LIN {X 0,Y 372.222,Z 970.071,A -85,B 0,C 180,E1 15608.829,E2 15608.829} C_VEL
LIN {X 0,Y 365.379,Z 983.592,A -85,B 0,C 180,E1 15606.041,E2 15606.041} C_VEL
LIN {X 0,Y 359.083,Z 996.112,A -85,B 0,C 180,E1 15603.054,E2 15603.054} C_VEL
LIN {X 0,Y 352.099,Z 1010.25,A -85,B 0,C 180,E1 15599.052,E2 15599.052} C_VEL
LIN {X 0,Y 347.306,Z 1020.442,A -85,B 0,C 180,E1 15595.585,E2 15595.585} C_VEL
LIN {X 0,Y 343.315,Z 1029.671,A -85,B 0,C 180,E1 15591.888,E2 15591.888} C_VEL
LIN {X 0,Y 339.875,Z 1038.664,A -85,B 0,C 180,E1 15587.462,E2 15587.462} C_VEL
LIN {X 0,Y 337.952,Z 1044.795,A -85,B 0,C 180,E1 15583.691,E2 15583.691} C_VEL
LIN {X 0,Y 336.82,Z 1049.482,A -85,B 0,C 180,E1 15580.087,E2 15580.087} C_VEL
LIN {X 0,Y 336.14,Z 1053.645,A -85,B 0,C 180,E1 15575.805,E2 15575.805} C_VEL
LIN {X 0,Y 335.934,Z 1055.971,A -85,B 0,C 180,E1 15571.876,E2 15571.876} C_VEL
LIN {X 0,Y 335.909,Z 1056.968,A -85,B 0,C 180,E1 15568.635,E2 15568.635} C_VEL
LIN {X 0,Y 335.91,Z 1057.084,A -85,B 0,C 180,E1 15565.39,E2 15565.39} C_VEL
LIN {X 0,Y 335.94,Z 1056.315,A -85,B 0,C 180,E1 15562.131,E2 15562.131} C_VEL
LIN {X 0,Y 336.1,Z 1054.654,A -85,B 0,C 180,E1 15558.85,E2 15558.85} C_VEL
LIN {X 0,Y 336.529,Z 1051.925,A -85,B 0,C 180,E1 15555.372,E2 15555.372} C_VEL
LIN {X 0,Y 337.552,Z 1047.758,A -85,B 0,C 180,E1 15551.521,E2 15551.521} C_VEL
LIN {X 0,Y 339.699,Z 1041.098,A -85,B 0,C 180,E1 15546.953,E2 15546.953} C_VEL
LIN {X 0,Y 342.404,Z 1034.312,A -85,B 0,C 180,E1 15543.275,E2 15543.275} C_VEL
LIN {X 0,Y 346.076,Z 1026.246,A -85,B 0,C 180,E1 15539.628,E2 15539.628} C_VEL
LIN {X 0,Y 352.06,Z 1014.26,A -85,B 0,C 180,E1 15535.19,E2 15535.19} C_VEL
LIN {X 0,Y 357.776,Z 1003.409,A -85,B 0,C 180,E1 15531.856,E2 15531.856} C_VEL
LIN {X 0,Y 365.253,Z 989.805,A -85,B 0,C 180,E1 15528.301,E2 15528.301} C_VEL
LIN {X 0,Y 368.811,Z 983.139,A -85,B 0,C 180,E1 15526.799,E2 15526.799} C_VEL
LIN {X 0,Y 370.327,Z 979.107,A -85,B 0,C 180,E1 15525.802,E2 15525.802} C_VEL
LIN {X 0,Y 371.602,Z 968.39,A -85,B 0,C 180,E1 15522.974,E2 15522.974} C_VEL
LIN {X 0,Y 373.172,Z 964.471,A -85,B 0,C 180,E1 15522.181,E2 15522.181} C_VEL
LIN {X 0,Y 381.333,Z 949.488,A -85,B 0,C 180,E1 15519.689,E2 15519.689} C_VEL
LIN {X 0,Y 390.212,Z 932.645,A -85,B 0,C 180,E1 15517.285,E2 15517.285} C_VEL
LIN {X 0,Y 400.258,Z 912.27,A -85,B 0,C 180,E1 15514.852,E2 15514.852} C_VEL
LIN {X 0,Y 408.245,Z 894.982,A -85,B 0,C 180,E1 15513.106,E2 15513.106} C_VEL
LIN {X 0,Y 416.573,Z 875.657,A -85,B 0,C 180,E1 15511.428,E2 15511.428} C_VEL
LIN {X 0,Y 425.589,Z 852.408,A -85,B 0,C 180,E1 15509.747,E2 15509.747} C_VEL
LIN {X 0,Y 432.181,Z 833.489,A -85,B 0,C 180,E1 15508.598,E2 15508.598} C_VEL
LIN {X 0,Y 438.616,Z 812.853,A -85,B 0,C 180,E1 15507.529,E2 15507.529} C_VEL
LIN {X 0,Y 445.749,Z 786.165,A -85,B 0,C 180,E1 15506.41,E2 15506.41} C_VEL
LIN {X 0,Y 450.602,Z 764.172,A -85,B 0,C 180,E1 15505.676,E2 15505.676} C_VEL
LIN {X 0,Y 454.876,Z 740.778,A -85,B 0,C 180,E1 15505.063,E2 15505.063} C_VEL
LIN {X 0,Y 458.362,Z 713.784,A -85,B 0,C 180,E1 15504.527,E2 15504.527} C_VEL
LIN {X 0,Y 473.41,Z 521.073,A -85,B 0,C 180,E1 15501.495,E2 15501.495} C_VEL
LIN {X 0,Y 477.59,Z 467.874,A -85,B 0,C 180,E1 15500.657,E2 15500.657} C_VEL
LIN {X 0,Y 470.268,Z 455.931,A -85,B 0,C 180,E1 15497.829,E2 15497.829} C_VEL
LIN {X 0,Y 464.119,Z 446.543,A -85,B 0,C 180,E1 15495.047,E2 15495.047} C_VEL
LIN {X 0,Y 460.67,Z 441.475,A -85,B 0,C 180,E1 15493.238,E2 15493.238} C_VEL
LIN {X 0,Y 457.903,Z 437.421,A -85,B 0,C 180,E1 15491.589,E2 15491.589} C_VEL
LIN {X 0,Y 454.898,Z 432.925,A -85,B 0,C 180,E1 15489.489,E2 15489.489} C_VEL
LIN {X 0,Y 451.914,Z 428.441,A -85,B 0,C 180,E1 15486.862,E2 15486.862} C_VEL
LIN {X 0,Y 448.733,Z 423.885,A -85,B 0,C 180,E1 15482.426,E2 15482.426} C_VEL
LIN {X 0,Y 448.35,Z 422.762,A -85,B 0,C 180,E1 15481.278,E2 15481.278} C_VEL
LIN {X 0,Y 448.16,Z 422.66,A -85,B 0,C 180,E1 15476.418,E2 15476.418} C_VEL
LIN {X 0,Y 448.576,Z 423.232,A -85,B 0,C 180,E1 15475.141,E2 15475.141} C_VEL
LIN {X 0,Y 450.853,Z 427.461,A -85,B 0,C 180,E1 15471.326,E2 15471.326} C_VEL
LIN {X 0,Y 452.07,Z 428.734,A -85,B 0,C 180,E1 15470.066,E2 15470.066} C_VEL
LIN {X 0,Y 455.617,Z 434.006,A -85,B 0,C 180,E1 15467.065,E2 15467.065} C_VEL
LIN {X 0,Y 459.489,Z 439.662,A -85,B 0,C 180,E1 15464.54,E2 15464.54} C_VEL
LIN {X 0,Y 462.897,Z 444.822,A -85,B 0,C 180,E1 15462.657,E2 15462.657} C_VEL
LIN {X 0,Y 467.926,Z 452.369,A -85,B 0,C 180,E1 15460.268,E2 15460.268} C_VEL
LIN {X 0,Y 473.578,Z 462.229,A -85,B 0,C 180,E1 15457.892,E2 15457.892} C_VEL
LIN {X 0,Y 477.55,Z 469.616,A -85,B 0,C 180,E1 15456.38,E2 15456.38} C_VEL
LIN {X 0,Y 459.798,Z 699.014,A -85,B 0,C 180,E1 15452.792,E2 15452.792} C_VEL
LIN {X 0,Y 456.746,Z 730.026,A -85,B 0,C 180,E1 15452.255,E2 15452.255} C_VEL
LIN {X 0,Y 453.419,Z 751.939,A -85,B 0,C 180,E1 15451.778,E2 15451.778} C_VEL
LIN {X 0,Y 448.791,Z 775.796,A -85,B 0,C 180,E1 15451.123,E2 15451.123} C_VEL
LIN {X 0,Y 442.754,Z 800.711,A -85,B 0,C 180,E1 15450.229,E2 15450.229} C_VEL
LIN {X 0,Y 436.754,Z 821.884,A -85,B 0,C 180,E1 15449.29,E2 15449.29} C_VEL
LIN {X 0,Y 429.461,Z 844.642,A -85,B 0,C 180,E1 15448.077,E2 15448.077} C_VEL
LIN {X 0,Y 421,Z 867.55,A -85,B 0,C 180,E1 15446.585,E2 15446.585} C_VEL
LIN {X 0,Y 413.553,Z 885.936,A -85,B 0,C 180,E1 15445.169,E2 15445.169} C_VEL
LIN {X 0,Y 404.883,Z 905.797,A -85,B 0,C 180,E1 15443.38,E2 15443.38} C_VEL
LIN {X 0,Y 395.21,Z 926.087,A -85,B 0,C 180,E1 15441.191,E2 15441.191} C_VEL
LIN {X 0,Y 387.162,Z 942.019,A -85,B 0,C 180,E1 15439.174,E2 15439.174} C_VEL
LIN {X 0,Y 378.632,Z 958.248,A -85,B 0,C 180,E1 15436.791,E2 15436.791} C_VEL
LIN {X 0,Y 368.644,Z 976.469,A -85,B 0,C 180,E1 15433.598,E2 15433.598} C_VEL
LIN {X 0,Y 361.117,Z 989.91,A -85,B 0,C 180,E1 15430.802,E2 15430.802} C_VEL
LIN {X 0,Y 353.453,Z 1003.67,A -85,B 0,C 180,E1 15427.461,E2 15427.461} C_VEL
LIN {X 0,Y 346.006,Z 1017.147,A -85,B 0,C 180,E1 15423.501,E2 15423.501} C_VEL
LIN {X 0,Y 340.806,Z 1027.013,A -85,B 0,C 180,E1 15420.06,E2 15420.06} C_VEL
LIN {X 0,Y 335.835,Z 1037.363,A -85,B 0,C 180,E1 15415.765,E2 15415.765} C_VEL
LIN {X 0,Y 332.319,Z 1045.488,A -85,B 0,C 180,E1 15411.535,E2 15411.535} C_VEL
LIN {X 0,Y 330.223,Z 1051.354,A -85,B 0,C 180,E1 15407.807,E2 15407.807} C_VEL
LIN {X 0,Y 328.785,Z 1056.688,A -85,B 0,C 180,E1 15403.543,E2 15403.543} C_VEL
LIN {X 0,Y 328.091,Z 1060.541,A -85,B 0,C 180,E1 15399.095,E2 15399.095} C_VEL
LIN {X 0,Y 327.924,Z 1062.495,A -85,B 0,C 180,E1 15395.599,E2 15395.599} C_VEL
LIN {X 0,Y 327.91,Z 1063.451,A -85,B 0,C 180,E1 15392.272,E2 15392.272} C_VEL
LIN {X 0,Y 327.914,Z 1063.508,A -85,B 0,C 180,E1 15388.952,E2 15388.952} C_VEL
LIN {X 0,Y 327.909,Z 1062.672,A -85,B 0,C 180,E1 15385.652,E2 15385.652} C_VEL
LIN {X 0,Y 328.019,Z 1060.834,A -85,B 0,C 180,E1 15382.177,E2 15382.177} C_VEL
LIN {X 0,Y 328.377,Z 1057.75,A -85,B 0,C 180,E1 15378.407,E2 15378.407} C_VEL
LIN {X 0,Y 329.528,Z 1052.362,A -85,B 0,C 180,E1 15373.79,E2 15373.79} C_VEL
LIN {X 0,Y 331.318,Z 1046.309,A -85,B 0,C 180,E1 15369.877,E2 15369.877} C_VEL
LIN {X 0,Y 333.901,Z 1039.288,A -85,B 0,C 180,E1 15366.155,E2 15366.155} C_VEL
LIN {X 0,Y 338.231,Z 1029.2,A -85,B 0,C 180,E1 15361.759,E2 15361.759} C_VEL
LIN {X 0,Y 343.228,Z 1018.544,A -85,B 0,C 180,E1 15357.967,E2 15357.967} C_VEL
LIN {X 0,Y 348.774,Z 1007.481,A -85,B 0,C 180,E1 15354.613,E2 15354.613} C_VEL
LIN {X 0,Y 356.78,Z 991.95,A -85,B 0,C 180,E1 15350.67,E2 15350.67} C_VEL
LIN {X 0,Y 363.591,Z 978.783,A -85,B 0,C 180,E1 15347.855,E2 15347.855} C_VEL
LIN {X 0,Y 371.311,Z 963.786,A -85,B 0,C 180,E1 15345.091,E2 15345.091} C_VEL
LIN {X 0,Y 380.835,Z 944.665,A -85,B 0,C 180,E1 15342.129,E2 15342.129} C_VEL
LIN {X 0,Y 388.709,Z 928.097,A -85,B 0,C 180,E1 15339.955,E2 15339.955} C_VEL
LIN {X 0,Y 397.375,Z 909.005,A -85,B 0,C 180,E1 15337.806,E2 15337.806} C_VEL
LIN {X 0,Y 406.238,Z 887.742,A -85,B 0,C 180,E1 15335.806,E2 15335.806} C_VEL
LIN {X 0,Y 413.53,Z 868.788,A -85,B 0,C 180,E1 15334.29,E2 15334.29} C_VEL
LIN {X 0,Y 421.537,Z 846.152,A -85,B 0,C 180,E1 15332.755,E2 15332.755} C_VEL
LIN {X 0,Y 428.551,Z 823.276,A -85,B 0,C 180,E1 15331.485,E2 15331.485} C_VEL
LIN {X 0,Y 434.162,Z 802.68,A -85,B 0,C 180,E1 15330.534,E2 15330.534} C_VEL
LIN {X 0,Y 439.741,Z 779.136,A -85,B 0,C 180,E1 15329.639,E2 15329.639} C_VEL
LIN {X 0,Y 444.546,Z 753.667,A -85,B 0,C 180,E1 15328.891,E2 15328.891} C_VEL
LIN {X 0,Y 447.739,Z 732.026,A -85,B 0,C 180,E1 15328.396,E2 15328.396} C_VEL
LIN {X 0,Y 450.405,Z 705.719,A -85,B 0,C 180,E1 15327.914,E2 15327.914} C_VEL
LIN {X 0,Y 467.057,Z 475.799,A -85,B 0,C 180,E1 15324.273,E2 15324.273} C_VEL
LIN {X 0,Y 467.908,Z 463.298,A -85,B 0,C 180,E1 15324.056,E2 15324.056} C_VEL
LIN {X 0,Y 460.162,Z 449.288,A -85,B 0,C 180,E1 15321.411,E2 15321.411} C_VEL
LIN {X 0,Y 456.588,Z 443.345,A -85,B 0,C 180,E1 15320.076,E2 15320.076} C_VEL
LIN {X 0,Y 449.632,Z 432.824,A -85,B 0,C 180,E1 15317.204,E2 15317.204} C_VEL
LIN {X 0,Y 444.966,Z 426.231,A -85,B 0,C 180,E1 15314.976,E2 15314.976} C_VEL
LIN {X 0,Y 442.403,Z 422.572,A -85,B 0,C 180,E1 15313.595,E2 15313.595} C_VEL
LIN {X 0,Y 439.27,Z 418.075,A -85,B 0,C 180,E1 15311.688,E2 15311.688} C_VEL
LIN {X 0,Y 435.894,Z 413.285,A -85,B 0,C 180,E1 15309.24,E2 15309.24} C_VEL
LIN {X 0,Y 432.824,Z 409.127,A -85,B 0,C 180,E1 15306.366,E2 15306.366} C_VEL
LIN {X 0,Y 432.182,Z 407.943,A -85,B 0,C 180,E1 15305.576,E2 15305.576} C_VEL
LIN {X 0,Y 429.28,Z 404.339,A -85,B 0,C 180,E1 15298.932,E2 15298.932} C_VEL
LIN {X 0,Y 429.455,Z 404.92,A -85,B 0,C 180,E1 15296.396,E2 15296.396} C_VEL
LIN {X 0,Y 432.483,Z 408.294,A -85,B 0,C 180,E1 15290.888,E2 15290.888} C_VEL
LIN {X 0,Y 435.038,Z 412.43,A -85,B 0,C 180,E1 15288.268,E2 15288.268} C_VEL
LIN {X 0,Y 436.506,Z 414.151,A -85,B 0,C 180,E1 15287.095,E2 15287.095} C_VEL
LIN {X 0,Y 440.335,Z 419.521,A -85,B 0,C 180,E1 15284.458,E2 15284.458} C_VEL
LIN {X 0,Y 444.324,Z 425.298,A -85,B 0,C 180,E1 15282.179,E2 15282.179} C_VEL
LIN {X 0,Y 448.509,Z 431.25,A -85,B 0,C 180,E1 15280.124,E2 15280.124} C_VEL
LIN {X 0,Y 453.666,Z 438.935,A -85,B 0,C 180,E1 15277.893,E2 15277.893} C_VEL
LIN {X 0,Y 461.118,Z 450.358,A -85,B 0,C 180,E1 15275.089,E2 15275.089} C_VEL
LIN {X 0,Y 468.016,Z 461.86,A -85,B 0,C 180,E1 15272.786,E2 15272.786} C_VEL
LIN {X 0,Y 451.586,Z 687.773,A -85,B 0,C 180,E1 15269.211,E2 15269.211} C_VEL
LIN {X 0,Y 448.571,Z 722.956,A -85,B 0,C 180,E1 15268.611,E2 15268.611} C_VEL
LIN {X 0,Y 445.268,Z 746.42,A -85,B 0,C 180,E1 15268.084,E2 15268.084} C_VEL
LIN {X 0,Y 441.55,Z 767.105,A -85,B 0,C 180,E1 15267.499,E2 15267.499} C_VEL
LIN {X 0,Y 436.014,Z 792.502,A -85,B 0,C 180,E1 15266.588,E2 15266.588} C_VEL
LIN {X 0,Y 429.88,Z 815.6,A -85,B 0,C 180,E1 15265.543,E2 15265.543} C_VEL
LIN {X 0,Y 423.603,Z 836.487,A -85,B 0,C 180,E1 15264.406,E2 15264.406} C_VEL
LIN {X 0,Y 415.065,Z 861.431,A -85,B 0,C 180,E1 15262.766,E2 15262.766} C_VEL
LIN {X 0,Y 407.73,Z 880.656,A -85,B 0,C 180,E1 15261.246,E2 15261.246} C_VEL
LIN {X 0,Y 400.217,Z 898.909,A -85,B 0,C 180,E1 15259.568,E2 15259.568} C_VEL
LIN {X 0,Y 390.481,Z 920.716,A -85,B 0,C 180,E1 15257.191,E2 15257.191} C_VEL
LIN {X 0,Y 382.696,Z 937.076,A -85,B 0,C 180,E1 15255.077,E2 15255.077} C_VEL
LIN {X 0,Y 374.725,Z 953.169,A -85,B 0,C 180,E1 15252.668,E2 15252.668} C_VEL
LIN {X 0,Y 365.636,Z 970.804,A -85,B 0,C 180,E1 15249.54,E2 15249.54} C_VEL
LIN {X 0,Y 358.424,Z 984.535,A -85,B 0,C 180,E1 15246.654,E2 15246.654} C_VEL
LIN {X 0,Y 351.335,Z 998.149,A -85,B 0,C 180,E1 15243.317,E2 15243.317} C_VEL
LIN {X 0,Y 344.432,Z 1011.473,A -85,B 0,C 180,E1 15239.38,E2 15239.38} C_VEL
LIN {X 0,Y 339.726,Z 1021.088,A -85,B 0,C 180,E1 15236.01,E2 15236.01} C_VEL
LIN {X 0,Y 335.266,Z 1031.048,A -85,B 0,C 180,E1 15231.888,E2 15231.888} C_VEL
LIN {X 0,Y 331.896,Z 1039.417,A -85,B 0,C 180,E1 15227.533,E2 15227.533} C_VEL
LIN {X 0,Y 330.01,Z 1045.188,A -85,B 0,C 180,E1 15223.849,E2 15223.849} C_VEL
LIN {X 0,Y 328.755,Z 1050.241,A -85,B 0,C 180,E1 15219.791,E2 15219.791} C_VEL
LIN {X 0,Y 328.099,Z 1054.199,A -85,B 0,C 180,E1 15215.246,E2 15215.246} C_VEL
LIN {X 0,Y 327.932,Z 1056.133,A -85,B 0,C 180,E1 15211.747,E2 15211.747} C_VEL
LIN {X 0,Y 327.908,Z 1057.051,A -85,B 0,C 180,E1 15208.602,E2 15208.602} C_VEL
LIN {X 0,Y 327.91,Z 1057.156,A -85,B 0,C 180,E1 15205.277,E2 15205.277} C_VEL
LIN {X 0,Y 327.947,Z 1056.377,A -85,B 0,C 180,E1 15201.938,E2 15201.938} C_VEL
LIN {X 0,Y 328.122,Z 1054.704,A -85,B 0,C 180,E1 15198.576,E2 15198.576} C_VEL
LIN {X 0,Y 328.598,Z 1051.964,A -85,B 0,C 180,E1 15195.01,E2 15195.01} C_VEL
LIN {X 0,Y 329.774,Z 1047.58,A -85,B 0,C 180,E1 15190.885,E2 15190.885} C_VEL
LIN {X 0,Y 332.139,Z 1040.835,A -85,B 0,C 180,E1 15186.232,E2 15186.232} C_VEL
LIN {X 0,Y 335.097,Z 1033.95,A -85,B 0,C 180,E1 15182.451,E2 15182.451} C_VEL
LIN {X 0,Y 339.552,Z 1024.874,A -85,B 0,C 180,E1 15178.324,E2 15178.324} C_VEL
LIN {X 0,Y 345.423,Z 1013.694,A -85,B 0,C 180,E1 15174.217,E2 15174.217} C_VEL
LIN {X 0,Y 351.173,Z 1003.346,A -85,B 0,C 180,E1 15171.005,E2 15171.005} C_VEL
LIN {X 0,Y 358.991,Z 989.725,A -85,B 0,C 180,E1 15167.404,E2 15167.404} C_VEL
LIN {X 0,Y 367.523,Z 974.523,A -85,B 0,C 180,E1 15164.091,E2 15164.091} C_VEL
LIN {X 0,Y 373.172,Z 964.471,A -85,B 0,C 180,E1 15162.181,E2 15162.181} C_VEL
LIN {X 0,Y 374.969,Z 959.913,A -85,B 0,C 180,E1 15161.261,E2 15161.261} C_VEL
LIN {X 0,Y 377.255,Z 948.11,A -85,B 0,C 180,E1 15158.592,E2 15158.592} C_VEL
LIN {X 0,Y 379.117,Z 943.873,A -85,B 0,C 180,E1 15157.866,E2 15157.866} C_VEL
LIN {X 0,Y 388.86,Z 925.372,A -85,B 0,C 180,E1 15155.402,E2 15155.402} C_VEL
LIN {X 0,Y 397.575,Z 907.914,A -85,B 0,C 180,E1 15153.421,E2 15153.421} C_VEL
LIN {X 0,Y 407.528,Z 886.509,A -85,B 0,C 180,E1 15151.369,E2 15151.369} C_VEL
LIN {X 0,Y 415.872,Z 866.607,A -85,B 0,C 180,E1 15149.778,E2 15149.778} C_VEL
LIN {X 0,Y 423.196,Z 847.602,A -85,B 0,C 180,E1 15148.487,E2 15148.487} C_VEL
LIN {X 0,Y 431.263,Z 824.335,A -85,B 0,C 180,E1 15147.154,E2 15147.154} C_VEL
LIN {X 0,Y 438.075,Z 801.282,A -85,B 0,C 180,E1 15146.085,E2 15146.085} C_VEL
LIN {X 0,Y 443.071,Z 781.883,A -85,B 0,C 180,E1 15145.336,E2 15145.336} C_VEL
LIN {X 0,Y 448.124,Z 758.724,A -85,B 0,C 180,E1 15144.599,E2 15144.599} C_VEL
LIN {X 0,Y 452.62,Z 732.06,A -85,B 0,C 180,E1 15143.963,E2 15143.963} C_VEL
LIN {X 0,Y 455.289,Z 709.677,A -85,B 0,C 180,E1 15143.549,E2 15143.549} C_VEL
LIN {X 0,Y 473.563,Z 481.081,A -85,B 0,C 180,E1 15139.973,E2 15139.973} C_VEL
LIN {X 0,Y 474.139,Z 472.834,A -85,B 0,C 180,E1 15139.816,E2 15139.816} C_VEL
LIN {X 0,Y 468.072,Z 462.777,A -85,B 0,C 180,E1 15137.37,E2 15137.37} C_VEL
LIN {X 0,Y 462.277,Z 453.737,A -85,B 0,C 180,E1 15134.659,E2 15134.659} C_VEL
LIN {X 0,Y 459.029,Z 448.861,A -85,B 0,C 180,E1 15132.901,E2 15132.901} C_VEL
LIN {X 0,Y 456.528,Z 445.104,A -85,B 0,C 180,E1 15131.369,E2 15131.369} C_VEL
LIN {X 0,Y 453.586,Z 440.634,A -85,B 0,C 180,E1 15129.26,E2 15129.26} C_VEL
LIN {X 0,Y 450.69,Z 436.123,A -85,B 0,C 180,E1 15126.625,E2 15126.625} C_VEL
LIN {X 0,Y 447.796,Z 432.079,A -85,B 0,C 180,E1 15122.56,E2 15122.56} C_VEL
LIN {X 0,Y 447.374,Z 430.709,A -85,B 0,C 180,E1 15121.281,E2 15121.281} C_VEL
LIN {X 0,Y 447.152,Z 430.583,A -85,B 0,C 180,E1 15116.539,E2 15116.539} C_VEL
LIN {X 0,Y 447.551,Z 431.124,A -85,B 0,C 180,E1 15115.258,E2 15115.258} C_VEL
LIN {X 0,Y 449.77,Z 435.343,A -85,B 0,C 180,E1 15111.434,E2 15111.434} C_VEL
LIN {X 0,Y 450.903,Z 436.557,A -85,B 0,C 180,E1 15110.233,E2 15110.233} C_VEL
LIN {X 0,Y 454.378,Z 441.861,A -85,B 0,C 180,E1 15107.223,E2 15107.223} C_VEL
LIN {X 0,Y 457.993,Z 447.212,A -85,B 0,C 180,E1 15104.812,E2 15104.812} C_VEL
LIN {X 0,Y 461.329,Z 452.378,A -85,B 0,C 180,E1 15102.921,E2 15102.921} C_VEL
LIN {X 0,Y 466.328,Z 460.082,A -85,B 0,C 180,E1 15100.491,E2 15100.491} C_VEL
LIN {X 0,Y 471.964,Z 470.201,A -85,B 0,C 180,E1 15098.075,E2 15098.075} C_VEL
LIN {X 0,Y 474.167,Z 474.485,A -85,B 0,C 180,E1 15097.202,E2 15097.202} C_VEL
LIN {X 0,Y 456.024,Z 703.267,A -85,B 0,C 180,E1 15093.632,E2 15093.632} C_VEL
LIN {X 0,Y 453.099,Z 730.953,A -85,B 0,C 180,E1 15093.145,E2 15093.145} C_VEL
LIN {X 0,Y 449.706,Z 752.666,A -85,B 0,C 180,E1 15092.672,E2 15092.672} C_VEL
LIN {X 0,Y 444.778,Z 777.432,A -85,B 0,C 180,E1 15091.99,E2 15091.99} C_VEL
LIN {X 0,Y 438.531,Z 802.213,A -85,B 0,C 180,E1 15091.093,E2 15091.093} C_VEL
LIN {X 0,Y 432.55,Z 822.752,A -85,B 0,C 180,E1 15090.181,E2 15090.181} C_VEL
LIN {X 0,Y 424.883,Z 846.005,A -85,B 0,C 180,E1 15088.938,E2 15088.938} C_VEL
LIN {X 0,Y 416.627,Z 867.707,A -85,B 0,C 180,E1 15087.52,E2 15087.52} C_VEL
LIN {X 0,Y 409.116,Z 885.779,A -85,B 0,C 180,E1 15086.135,E2 15086.135} C_VEL
LIN {X 0,Y 400.062,Z 905.976,A -85,B 0,C 180,E1 15084.319,E2 15084.319} C_VEL
LIN {X 0,Y 390.116,Z 926.223,A -85,B 0,C 180,E1 15082.131,E2 15082.131} C_VEL
LIN {X 0,Y 381.676,Z 942.42,A -85,B 0,C 180,E1 15080.071,E2 15080.071} C_VEL
LIN {X 0,Y 372.528,Z 959.268,A -85,B 0,C 180,E1 15077.571,E2 15077.571} C_VEL
LIN {X 0,Y 362.578,Z 976.723,A -85,B 0,C 180,E1 15074.464,E2 15074.464} C_VEL
LIN {X 0,Y 354.872,Z 989.964,A -85,B 0,C 180,E1 15071.679,E2 15071.679} C_VEL
LIN {X 0,Y 346.886,Z 1003.71,A -85,B 0,C 180,E1 15068.296,E2 15068.296} C_VEL
LIN {X 0,Y 339.313,Z 1016.791,A -85,B 0,C 180,E1 15064.4,E2 15064.4} C_VEL
LIN {X 0,Y 333.949,Z 1026.437,A -85,B 0,C 180,E1 15060.997,E2 15060.997} C_VEL
LIN {X 0,Y 329.145,Z 1035.776,A -85,B 0,C 180,E1 15057.108,E2 15057.108} C_VEL
LIN {X 0,Y 324.918,Z 1044.856,A -85,B 0,C 180,E1 15052.432,E2 15052.432} C_VEL
LIN {X 0,Y 322.59,Z 1050.81,A -85,B 0,C 180,E1 15048.618,E2 15048.618} C_VEL
LIN {X 0,Y 321.111,Z 1055.607,A -85,B 0,C 180,E1 15044.793,E2 15044.793} C_VEL
LIN {X 0,Y 320.207,Z 1059.893,A -85,B 0,C 180,E1 15040.253,E2 15040.253} C_VEL
LIN {X 0,Y 319.939,Z 1062.291,A -85,B 0,C 180,E1 15036.1,E2 15036.1} C_VEL
LIN {X 0,Y 319.913,Z 1063.354,A -85,B 0,C 180,E1 15032.508,E2 15032.508} C_VEL
LIN {X 0,Y 319.914,Z 1063.449,A -85,B 0,C 180,E1 15029.105,E2 15029.105} C_VEL
LIN {X 0,Y 319.91,Z 1062.642,A -85,B 0,C 180,E1 15025.698,E2 15025.698} C_VEL
LIN {X 0,Y 320.012,Z 1060.926,A -85,B 0,C 180,E1 15022.279,E2 15022.279} C_VEL
LIN {X 0,Y 320.355,Z 1058.021,A -85,B 0,C 180,E1 15018.539,E2 15018.539} C_VEL
LIN {X 0,Y 321.412,Z 1053.248,A -85,B 0,C 180,E1 15014.112,E2 15014.112} C_VEL
LIN {X 0,Y 323.37,Z 1046.788,A -85,B 0,C 180,E1 15009.738,E2 15009.738} C_VEL
LIN {X 0,Y 326.029,Z 1039.857,A -85,B 0,C 180,E1 15005.928,E2 15005.928} C_VEL
LIN {X 0,Y 330.07,Z 1030.828,A -85,B 0,C 180,E1 15001.799,E2 15001.799} C_VEL
LIN {X 0,Y 335.632,Z 1019.444,A -85,B 0,C 180,E1 14997.572,E2 14997.572} C_VEL
LIN {X 0,Y 341.064,Z 1009.003,A -85,B 0,C 180,E1 14994.3,E2 14994.3} C_VEL
LIN {X 0,Y 348.464,Z 995.34,A -85,B 0,C 180,E1 14990.644,E2 14990.644} C_VEL
LIN {X 0,Y 356.608,Z 980.113,A -85,B 0,C 180,E1 14987.271,E2 14987.271} C_VEL
LIN {X 0,Y 363.993,Z 966.255,A -85,B 0,C 180,E1 14984.646,E2 14984.646} C_VEL
LIN {X 0,Y 373.309,Z 948.461,A -85,B 0,C 180,E1 14981.76,E2 14981.76} C_VEL
LIN {X 0,Y 382.499,Z 929.747,A -85,B 0,C 180,E1 14979.243,E2 14979.243} C_VEL
LIN {X 0,Y 390.347,Z 912.993,A -85,B 0,C 180,E1 14977.312,E2 14977.312} C_VEL
LIN {X 0,Y 399.68,Z 891.819,A -85,B 0,C 180,E1 14975.231,E2 14975.231} C_VEL
LIN {X 0,Y 407.893,Z 871.174,A -85,B 0,C 180,E1 14973.545,E2 14973.545} C_VEL
LIN {X 0,Y 414.854,Z 852.181,A -85,B 0,C 180,E1 14972.223,E2 14972.223} C_VEL
LIN {X 0,Y 422.698,Z 828.468,A -85,B 0,C 180,E1 14970.833,E2 14970.833} C_VEL
LIN {X 0,Y 429.139,Z 805.721,A -85,B 0,C 180,E1 14969.755,E2 14969.755} C_VEL
LIN {X 0,Y 434.043,Z 785.947,A -85,B 0,C 180,E1 14968.977,E2 14968.977} C_VEL
LIN {X 0,Y 438.78,Z 763.455,A -85,B 0,C 180,E1 14968.249,E2 14968.249} C_VEL
LIN {X 0,Y 443.219,Z 736.393,A -85,B 0,C 180,E1 14967.587,E2 14967.587} C_VEL
LIN {X 0,Y 445.776,Z 713.951,A -85,B 0,C 180,E1 14967.159,E2 14967.159} C_VEL
LIN {X 0,Y 462.831,Z 486.295,A -85,B 0,C 180,E1 14963.546,E2 14963.546} C_VEL
LIN {X 0,Y 464.212,Z 467.843,A -85,B 0,C 180,E1 14963.248,E2 14963.248} C_VEL
LIN {X 0,Y 455.965,Z 452.756,A -85,B 0,C 180,E1 14960.272,E2 14960.272} C_VEL
LIN {X 0,Y 448.889,Z 441.9,A -85,B 0,C 180,E1 14957.367,E2 14957.367} C_VEL
LIN {X 0,Y 443.848,Z 434.451,A -85,B 0,C 180,E1 14954.948,E2 14954.948} C_VEL
LIN {X 0,Y 440.745,Z 429.971,A -85,B 0,C 180,E1 14953.246,E2 14953.246} C_VEL
LIN {X 0,Y 437.792,Z 425.655,A -85,B 0,C 180,E1 14951.394,E2 14951.394} C_VEL
LIN {X 0,Y 434.586,Z 421.013,A -85,B 0,C 180,E1 14949.001,E2 14949.001} C_VEL
LIN {X 0,Y 431.614,Z 416.809,A -85,B 0,C 180,E1 14946.117,E2 14946.117} C_VEL
LIN {X 0,Y 431.094,Z 415.835,A -85,B 0,C 180,E1 14945.457,E2 14945.457} C_VEL
LIN {X 0,Y 428.3,Z 412.255,A -85,B 0,C 180,E1 14938.796,E2 14938.796} C_VEL
LIN {X 0,Y 428.506,Z 412.956,A -85,B 0,C 180,E1 14936.254,E2 14936.254} C_VEL
LIN {X 0,Y 431.389,Z 416.248,A -85,B 0,C 180,E1 14930.999,E2 14930.999} C_VEL
LIN {X 0,Y 433.997,Z 420.407,A -85,B 0,C 180,E1 14928.302,E2 14928.302} C_VEL
LIN {X 0,Y 435.275,Z 422.004,A -85,B 0,C 180,E1 14927.26,E2 14927.26} C_VEL
LIN {X 0,Y 439.042,Z 427.417,A -85,B 0,C 180,E1 14924.614,E2 14924.614} C_VEL
LIN {X 0,Y 442.749,Z 432.855,A -85,B 0,C 180,E1 14922.453,E2 14922.453} C_VEL
LIN {X 0,Y 446.859,Z 438.811,A -85,B 0,C 180,E1 14920.388,E2 14920.388} C_VEL
LIN {X 0,Y 452.372,Z 447.242,A -85,B 0,C 180,E1 14917.963,E2 14917.963} C_VEL
LIN {X 0,Y 459.03,Z 457.673,A -85,B 0,C 180,E1 14915.414,E2 14915.414} C_VEL
LIN {X 0,Y 464.259,Z 466.549,A -85,B 0,C 180,E1 14913.606,E2 14913.606} C_VEL
LIN {X 0,Y 447.312,Z 693.706,A -85,B 0,C 180,E1 14910.014,E2 14910.014} C_VEL
LIN {X 0,Y 444.301,Z 725.671,A -85,B 0,C 180,E1 14909.454,E2 14909.454} C_VEL
LIN {X 0,Y 441.078,Z 747.714,A -85,B 0,C 180,E1 14908.953,E2 14908.953} C_VEL
LIN {X 0,Y 437.082,Z 769.265,A -85,B 0,C 180,E1 14908.336,E2 14908.336} C_VEL
LIN {X 0,Y 431.01,Z 795.712,A -85,B 0,C 180,E1 14907.363,E2 14907.363} C_VEL
LIN {X 0,Y 425.408,Z 816.204,A -85,B 0,C 180,E1 14906.431,E2 14906.431} C_VEL
LIN {X 0,Y 418.992,Z 837.035,A -85,B 0,C 180,E1 14905.297,E2 14905.297} C_VEL
LIN {X 0,Y 410.249,Z 861.89,A -85,B 0,C 180,E1 14903.66,E2 14903.66} C_VEL
LIN {X 0,Y 402.732,Z 881.08,A -85,B 0,C 180,E1 14902.14,E2 14902.14} C_VEL
LIN {X 0,Y 394.641,Z 900.191,A -85,B 0,C 180,E1 14900.375,E2 14900.375} C_VEL
LIN {X 0,Y 385.014,Z 921.061,A -85,B 0,C 180,E1 14898.077,E2 14898.077} C_VEL
LIN {X 0,Y 376.996,Z 937.399,A -85,B 0,C 180,E1 14895.952,E2 14895.952} C_VEL
LIN {X 0,Y 368.307,Z 954.386,A -85,B 0,C 180,E1 14893.381,E2 14893.381} C_VEL
LIN {X 0,Y 359.029,Z 971.677,A -85,B 0,C 180,E1 14890.249,E2 14890.249} C_VEL
LIN {X 0,Y 351.885,Z 984.787,A -85,B 0,C 180,E1 14887.451,E2 14887.451} C_VEL
LIN {X 0,Y 344.514,Z 998.385,A -85,B 0,C 180,E1 14884.066,E2 14884.066} C_VEL
LIN {X 0,Y 337.586,Z 1011.172,A -85,B 0,C 180,E1 14880.233,E2 14880.233} C_VEL
LIN {X 0,Y 332.528,Z 1020.996,A -85,B 0,C 180,E1 14876.739,E2 14876.739} C_VEL
LIN {X 0,Y 327.865,Z 1030.83,A -85,B 0,C 180,E1 14872.598,E2 14872.598} C_VEL
LIN {X 0,Y 324.265,Z 1039.272,A -85,B 0,C 180,E1 14868.146,E2 14868.146} C_VEL
LIN {X 0,Y 322.224,Z 1045.079,A -85,B 0,C 180,E1 14864.374,E2 14864.374} C_VEL
LIN {X 0,Y 320.894,Z 1049.946,A -85,B 0,C 180,E1 14860.412,E2 14860.412} C_VEL
LIN {X 0,Y 320.137,Z 1054.081,A -85,B 0,C 180,E1 14855.736,E2 14855.736} C_VEL
LIN {X 0,Y 319.937,Z 1056.161,A -85,B 0,C 180,E1 14851.97,E2 14851.97} C_VEL
LIN {X 0,Y 319.908,Z 1057.135,A -85,B 0,C 180,E1 14848.567,E2 14848.567} C_VEL
LIN {X 0,Y 319.911,Z 1057.229,A -85,B 0,C 180,E1 14845.159,E2 14845.159} C_VEL
LIN {X 0,Y 319.957,Z 1056.438,A -85,B 0,C 180,E1 14841.735,E2 14841.735} C_VEL
LIN {X 0,Y 320.146,Z 1054.755,A -85,B 0,C 180,E1 14838.287,E2 14838.287} C_VEL
LIN {X 0,Y 320.676,Z 1052.003,A -85,B 0,C 180,E1 14834.631,E2 14834.631} C_VEL
LIN {X 0,Y 322.032,Z 1047.402,A -85,B 0,C 180,E1 14830.218,E2 14830.218} C_VEL
LIN {X 0,Y 324.529,Z 1040.802,A -85,B 0,C 180,E1 14825.615,E2 14825.615} C_VEL
LIN {X 0,Y 327.678,Z 1033.941,A -85,B 0,C 180,E1 14821.773,E2 14821.773} C_VEL
LIN {X 0,Y 332.576,Z 1024.576,A -85,B 0,C 180,E1 14817.441,E2 14817.441} C_VEL
LIN {X 0,Y 338.606,Z 1013.645,A -85,B 0,C 180,E1 14813.381,E2 14813.381} C_VEL
LIN {X 0,Y 344.657,Z 1003.283,A -85,B 0,C 180,E1 14810.123,E2 14810.123} C_VEL
LIN {X 0,Y 352.815,Z 989.642,A -85,B 0,C 180,E1 14806.475,E2 14806.475} C_VEL
LIN {X 0,Y 361.705,Z 974.412,A -85,B 0,C 180,E1 14803.131,E2 14803.131} C_VEL
LIN {X 0,Y 369.715,Z 960.563,A -85,B 0,C 180,E1 14800.54,E2 14800.54} C_VEL
LIN {X 0,Y 379.117,Z 943.873,A -85,B 0,C 180,E1 14797.866,E2 14797.866} C_VEL
LIN {X 0,Y 381.221,Z 938.872,A -85,B 0,C 180,E1 14797.029,E2 14797.029} C_VEL
LIN {X 0,Y 383.971,Z 926.574,A -85,B 0,C 180,E1 14794.682,E2 14794.682} C_VEL
LIN {X 0,Y 386.184,Z 921.228,A -85,B 0,C 180,E1 14793.911,E2 14793.911} C_VEL
LIN {X 0,Y 397.054,Z 899.548,A -85,B 0,C 180,E1 14791.588,E2 14791.588} C_VEL
LIN {X 0,Y 405.557,Z 881.046,A -85,B 0,C 180,E1 14789.933,E2 14789.933} C_VEL
LIN {X 0,Y 413.199,Z 863.024,A -85,B 0,C 180,E1 14788.549,E2 14788.549} C_VEL
LIN {X 0,Y 422.124,Z 839.799,A -85,B 0,C 180,E1 14787.047,E2 14787.047} C_VEL
LIN {X 0,Y 429.502,Z 817.652,A -85,B 0,C 180,E1 14785.871,E2 14785.871} C_VEL
LIN {X 0,Y 435.622,Z 796.863,A -85,B 0,C 180,E1 14784.954,E2 14784.954} C_VEL
LIN {X 0,Y 442.004,Z 771.305,A -85,B 0,C 180,E1 14784.042,E2 14784.042} C_VEL
LIN {X 0,Y 446.581,Z 748.346,A -85,B 0,C 180,E1 14783.408,E2 14783.408} C_VEL
LIN {X 0,Y 449.964,Z 726.824,A -85,B 0,C 180,E1 14782.936,E2 14782.936} C_VEL
LIN {X 0,Y 453,Z 698.241,A -85,B 0,C 180,E1 14782.439,E2 14782.439} C_VEL
LIN {X 0,Y 470.923,Z 477.978,A -85,B 0,C 180,E1 14779.013,E2 14779.013} C_VEL
LIN {X 0,Y 464.858,Z 467.908,A -85,B 0,C 180,E1 14776.431,E2 14776.431} C_VEL
LIN {X 0,Y 459.777,Z 459.859,A -85,B 0,C 180,E1 14773.905,E2 14773.905} C_VEL
LIN {X 0,Y 455.448,Z 453.141,A -85,B 0,C 180,E1 14771.332,E2 14771.332} C_VEL
LIN {X 0,Y 452.282,Z 448.342,A -85,B 0,C 180,E1 14769.031,E2 14769.031} C_VEL
LIN {X 0,Y 449.227,Z 443.618,A -85,B 0,C 180,E1 14766.133,E2 14766.133} C_VEL
LIN {X 0,Y 446.76,Z 439.956,A -85,B 0,C 180,E1 14762.437,E2 14762.437} C_VEL
LIN {X 0,Y 446.356,Z 438.616,A -85,B 0,C 180,E1 14761.155,E2 14761.155} C_VEL
LIN {X 0,Y 446.249,Z 438.567,A -85,B 0,C 180,E1 14756.274,E2 14756.274} C_VEL
LIN {X 0,Y 446.564,Z 439.185,A -85,B 0,C 180,E1 14755.248,E2 14755.248} C_VEL
LIN {X 0,Y 448.8,Z 443.33,A -85,B 0,C 180,E1 14751.415,E2 14751.415} C_VEL
LIN {X 0,Y 449.796,Z 444.505,A -85,B 0,C 180,E1 14750.338,E2 14750.338} C_VEL
LIN {X 0,Y 453.064,Z 449.562,A -85,B 0,C 180,E1 14747.444,E2 14747.444} C_VEL
LIN {X 0,Y 456.702,Z 455.094,A -85,B 0,C 180,E1 14744.963,E2 14744.963} C_VEL
LIN {X 0,Y 459.882,Z 460.114,A -85,B 0,C 180,E1 14743.126,E2 14743.126} C_VEL
LIN {X 0,Y 464.609,Z 467.569,A -85,B 0,C 180,E1 14740.775,E2 14740.775} C_VEL
LIN {X 0,Y 470.502,Z 478.416,A -85,B 0,C 180,E1 14738.2,E2 14738.2} C_VEL
LIN {X 0,Y 470.876,Z 479.45,A -85,B 0,C 180,E1 14738.034,E2 14738.034} C_VEL
LIN {X 0,Y 452.247,Z 708.25,A -85,B 0,C 180,E1 14734.471,E2 14734.471} C_VEL
LIN {X 0,Y 449.472,Z 732.529,A -85,B 0,C 180,E1 14734.037,E2 14734.037} C_VEL
LIN {X 0,Y 445.878,Z 754.693,A -85,B 0,C 180,E1 14733.55,E2 14733.55} C_VEL
LIN {X 0,Y 440.19,Z 781.577,A -85,B 0,C 180,E1 14732.784,E2 14732.784} C_VEL
LIN {X 0,Y 434.681,Z 802.749,A -85,B 0,C 180,E1 14732.014,E2 14732.014} C_VEL
LIN {X 0,Y 428.384,Z 823.838,A -85,B 0,C 180,E1 14731.078,E2 14731.078} C_VEL
LIN {X 0,Y 419.766,Z 848.883,A -85,B 0,C 180,E1 14729.721,E2 14729.721} C_VEL
LIN {X 0,Y 412.001,Z 868.751,A -85,B 0,C 180,E1 14728.413,E2 14728.413} C_VEL
LIN {X 0,Y 404.161,Z 887.08,A -85,B 0,C 180,E1 14727.001,E2 14727.001} C_VEL
LIN {X 0,Y 394.006,Z 908.921,A -85,B 0,C 180,E1 14725.003,E2 14725.003} C_VEL
LIN {X 0,Y 384.551,Z 927.463,A -85,B 0,C 180,E1 14722.962,E2 14722.962} C_VEL
LIN {X 0,Y 375.776,Z 943.766,A -85,B 0,C 180,E1 14720.863,E2 14720.863} C_VEL
LIN {X 0,Y 365.48,Z 962.026,A -85,B 0,C 180,E1 14718.085,E2 14718.085} C_VEL
LIN {X 0,Y 356.054,Z 977.875,A -85,B 0,C 180,E1 14715.181,E2 14715.181} C_VEL
LIN {X 0,Y 347.873,Z 991.416,A -85,B 0,C 180,E1 14712.267,E2 14712.267} C_VEL
LIN {X 0,Y 338.573,Z 1006.694,A -85,B 0,C 180,E1 14708.329,E2 14708.329} C_VEL
LIN {X 0,Y 331.945,Z 1017.695,A -85,B 0,C 180,E1 14704.912,E2 14704.912} C_VEL
LIN {X 0,Y 326.08,Z 1027.819,A -85,B 0,C 180,E1 14701.213,E2 14701.213} C_VEL
LIN {X 0,Y 320.216,Z 1038.749,A -85,B 0,C 180,E1 14696.321,E2 14696.321} C_VEL
LIN {X 0,Y 316.832,Z 1045.852,A -85,B 0,C 180,E1 14692.379,E2 14692.379} C_VEL
LIN {X 0,Y 314.44,Z 1051.798,A -85,B 0,C 180,E1 14688.349,E2 14688.349} C_VEL
LIN {X 0,Y 312.768,Z 1057.295,A -85,B 0,C 180,E1 14683.496,E2 14683.496} C_VEL
LIN {X 0,Y 312.112,Z 1060.558,A -85,B 0,C 180,E1 14679.348,E2 14679.348} C_VEL
LIN {X 0,Y 311.931,Z 1062.363,A -85,B 0,C 180,E1 14675.888,E2 14675.888} C_VEL
LIN {X 0,Y 311.911,Z 1063.303,A -85,B 0,C 180,E1 14672.389,E2 14672.389} C_VEL
LIN {X 0,Y 311.914,Z 1063.367,A -85,B 0,C 180,E1 14669.082,E2 14669.082} C_VEL
LIN {X 0,Y 311.91,Z 1062.552,A -85,B 0,C 180,E1 14665.588,E2 14665.588} C_VEL
LIN {X 0,Y 312.023,Z 1060.827,A -85,B 0,C 180,E1 14662.08,E2 14662.08} C_VEL
LIN {X 0,Y 312.379,Z 1058.02,A -85,B 0,C 180,E1 14658.366,E2 14658.366} C_VEL
LIN {X 0,Y 313.413,Z 1053.55,A -85,B 0,C 180,E1 14654.076,E2 14654.076} C_VEL
LIN {X 0,Y 315.533,Z 1046.959,A -85,B 0,C 180,E1 14649.406,E2 14649.406} C_VEL
LIN {X 0,Y 318.321,Z 1040.069,A -85,B 0,C 180,E1 14645.504,E2 14645.504} C_VEL
LIN {X 0,Y 322.329,Z 1031.491,A -85,B 0,C 180,E1 14641.464,E2 14641.464} C_VEL
LIN {X 0,Y 328.338,Z 1019.786,A -85,B 0,C 180,E1 14636.968,E2 14636.968} C_VEL
LIN {X 0,Y 334.301,Z 1008.842,A -85,B 0,C 180,E1 14633.473,E2 14633.473} C_VEL
LIN {X 0,Y 342.148,Z 994.946,A -85,B 0,C 180,E1 14629.707,E2 14629.707} C_VEL
LIN {X 0,Y 350.514,Z 979.881,A -85,B 0,C 180,E1 14626.344,E2 14626.344} C_VEL
LIN {X 0,Y 358.18,Z 966.009,A -85,B 0,C 180,E1 14623.696,E2 14623.696} C_VEL
LIN {X 0,Y 367.823,Z 948.186,A -85,B 0,C 180,E1 14620.794,E2 14620.794} C_VEL
LIN {X 0,Y 377.16,Z 929.748,A -85,B 0,C 180,E1 14618.305,E2 14618.305} C_VEL
LIN {X 0,Y 385.391,Z 912.674,A -85,B 0,C 180,E1 14616.334,E2 14616.334} C_VEL
LIN {X 0,Y 394.976,Z 891.465,A -85,B 0,C 180,E1 14614.256,E2 14614.256} C_VEL
LIN {X 0,Y 403.413,Z 870.777,A -85,B 0,C 180,E1 14612.573,E2 14612.573} C_VEL
LIN {X 0,Y 410.593,Z 851.604,A -85,B 0,C 180,E1 14611.246,E2 14611.246} C_VEL
LIN {X 0,Y 418.565,Z 827.942,A -85,B 0,C 180,E1 14609.871,E2 14609.871} C_VEL
LIN {X 0,Y 425.078,Z 805.408,A -85,B 0,C 180,E1 14608.812,E2 14608.812} C_VEL
LIN {X 0,Y 430.164,Z 785.288,A -85,B 0,C 180,E1 14608.03,E2 14608.03} C_VEL
LIN {X 0,Y 435.095,Z 762.276,A -85,B 0,C 180,E1 14607.297,E2 14607.297} C_VEL
LIN {X 0,Y 439.435,Z 735.953,A -85,B 0,C 180,E1 14606.664,E2 14606.664} C_VEL
LIN {X 0,Y 442.022,Z 713.611,A -85,B 0,C 180,E1 14606.241,E2 14606.241} C_VEL
LIN {X 0,Y 459.498,Z 486.235,A -85,B 0,C 180,E1 14602.638,E2 14602.638} C_VEL
LIN {X 0,Y 460.518,Z 472.293,A -85,B 0,C 180,E1 14602.399,E2 14602.399} C_VEL
LIN {X 0,Y 453.468,Z 459.299,A -85,B 0,C 180,E1 14599.75,E2 14599.75} C_VEL
LIN {X 0,Y 446.21,Z 447.811,A -85,B 0,C 180,E1 14596.635,E2 14596.635} C_VEL
LIN {X 0,Y 440.21,Z 438.755,A -85,B 0,C 180,E1 14593.53,E2 14593.53} C_VEL
LIN {X 0,Y 436.421,Z 433.343,A -85,B 0,C 180,E1 14591.163,E2 14591.163} C_VEL
LIN {X 0,Y 433.286,Z 428.738,A -85,B 0,C 180,E1 14588.761,E2 14588.761} C_VEL
LIN {X 0,Y 430.363,Z 424.37,A -85,B 0,C 180,E1 14585.801,E2 14585.801} C_VEL
LIN {X 0,Y 429.787,Z 423.595,A -85,B 0,C 180,E1 14585.072,E2 14585.072} C_VEL
LIN {X 0,Y 427.324,Z 420.197,A -85,B 0,C 180,E1 14578.793,E2 14578.793} C_VEL
LIN {X 0,Y 427.53,Z 420.918,A -85,B 0,C 180,E1 14576.245,E2 14576.245} C_VEL
LIN {X 0,Y 430.249,Z 424.071,A -85,B 0,C 180,E1 14571.177,E2 14571.177} C_VEL
LIN {X 0,Y 432.873,Z 428.295,A -85,B 0,C 180,E1 14568.407,E2 14568.407} C_VEL
LIN {X 0,Y 434.047,Z 429.853,A -85,B 0,C 180,E1 14567.426,E2 14567.426} C_VEL
LIN {X 0,Y 437.559,Z 434.968,A -85,B 0,C 180,E1 14564.9,E2 14564.9} C_VEL
LIN {X 0,Y 441.184,Z 440.411,A -85,B 0,C 180,E1 14562.729,E2 14562.729} C_VEL
LIN {X 0,Y 446.212,Z 447.748,A -85,B 0,C 180,E1 14560.188,E2 14560.188} C_VEL
LIN {X 0,Y 453.176,Z 458.883,A -85,B 0,C 180,E1 14557.184,E2 14557.184} C_VEL
LIN {X 0,Y 459.004,Z 468.453,A -85,B 0,C 180,E1 14555,E2 14555} C_VEL
LIN {X 0,Y 460.582,Z 471.467,A -85,B 0,C 180,E1 14554.434,E2 14554.434} C_VEL
LIN {X 0,Y 443.058,Z 700.569,A -85,B 0,C 180,E1 14550.818,E2 14550.818} C_VEL
LIN {X 0,Y 440.254,Z 727.454,A -85,B 0,C 180,E1 14550.332,E2 14550.332} C_VEL
LIN {X 0,Y 436.967,Z 749.146,A -85,B 0,C 180,E1 14549.836,E2 14549.836} C_VEL
LIN {X 0,Y 432.248,Z 773.755,A -85,B 0,C 180,E1 14549.115,E2 14549.115} C_VEL
LIN {X 0,Y 426.531,Z 797.244,A -85,B 0,C 180,E1 14548.229,E2 14548.229} C_VEL
LIN {X 0,Y 420.709,Z 817.921,A -85,B 0,C 180,E1 14547.282,E2 14547.282} C_VEL
LIN {X 0,Y 413.192,Z 841.529,A -85,B 0,C 180,E1 14545.977,E2 14545.977} C_VEL
LIN {X 0,Y 404.904,Z 863.952,A -85,B 0,C 180,E1 14544.457,E2 14544.457} C_VEL
LIN {X 0,Y 397.531,Z 882.231,A -85,B 0,C 180,E1 14542.995,E2 14542.995} C_VEL
LIN {X 0,Y 388.377,Z 903.193,A -85,B 0,C 180,E1 14541.032,E2 14541.032} C_VEL
LIN {X 0,Y 378.814,Z 923.047,A -85,B 0,C 180,E1 14538.786,E2 14538.786} C_VEL
LIN {X 0,Y 370.869,Z 938.721,A -85,B 0,C 180,E1 14536.713,E2 14536.713} C_VEL
LIN {X 0,Y 361.469,Z 956.483,A -85,B 0,C 180,E1 14533.972,E2 14533.972} C_VEL
LIN {X 0,Y 352.393,Z 972.704,A -85,B 0,C 180,E1 14530.953,E2 14530.953} C_VEL
LIN {X 0,Y 344.644,Z 986.419,A -85,B 0,C 180,E1 14527.956,E2 14527.956} C_VEL
LIN {X 0,Y 336.072,Z 1001.527,A -85,B 0,C 180,E1 14524.01,E2 14524.01} C_VEL
LIN {X 0,Y 329.963,Z 1012.393,A -85,B 0,C 180,E1 14520.603,E2 14520.603} C_VEL
LIN {X 0,Y 324.855,Z 1021.926,A -85,B 0,C 180,E1 14517.099,E2 14517.099} C_VEL
LIN {X 0,Y 319.809,Z 1032.097,A -85,B 0,C 180,E1 14512.616,E2 14512.616} C_VEL
LIN {X 0,Y 316.414,Z 1039.725,A -85,B 0,C 180,E1 14508.421,E2 14508.421} C_VEL
LIN {X 0,Y 314.293,Z 1045.472,A -85,B 0,C 180,E1 14504.556,E2 14504.556} C_VEL
LIN {X 0,Y 312.79,Z 1050.885,A -85,B 0,C 180,E1 14499.94,E2 14499.94} C_VEL
LIN {X 0,Y 312.122,Z 1054.412,A -85,B 0,C 180,E1 14495.515,E2 14495.515} C_VEL
LIN {X 0,Y 311.935,Z 1056.323,A -85,B 0,C 180,E1 14491.837,E2 14491.837} C_VEL
LIN {X 0,Y 311.908,Z 1057.218,A -85,B 0,C 180,E1 14488.53,E2 14488.53} C_VEL
LIN {X 0,Y 311.912,Z 1057.301,A -85,B 0,C 180,E1 14485.035,E2 14485.035} C_VEL
LIN {X 0,Y 311.965,Z 1056.5,A -85,B 0,C 180,E1 14481.522,E2 14481.522} C_VEL
LIN {X 0,Y 312.173,Z 1054.805,A -85,B 0,C 180,E1 14477.983,E2 14477.983} C_VEL
LIN {X 0,Y 312.772,Z 1052.023,A -85,B 0,C 180,E1 14474.209,E2 14474.209} C_VEL
LIN {X 0,Y 314.333,Z 1047.215,A -85,B 0,C 180,E1 14469.518,E2 14469.518} C_VEL
LIN {X 0,Y 317.041,Z 1040.568,A -85,B 0,C 180,E1 14464.844,E2 14464.844} C_VEL
LIN {X 0,Y 320.298,Z 1033.933,A -85,B 0,C 180,E1 14461.062,E2 14461.062} C_VEL
LIN {X 0,Y 325.501,Z 1024.551,A -85,B 0,C 180,E1 14456.643,E2 14456.643} C_VEL
LIN {X 0,Y 331.871,Z 1013.597,A -85,B 0,C 180,E1 14452.512,E2 14452.512} C_VEL
LIN {X 0,Y 338.291,Z 1003.105,A -85,B 0,C 180,E1 14449.171,E2 14449.171} C_VEL
LIN {X 0,Y 346.735,Z 989.556,A -85,B 0,C 180,E1 14445.513,E2 14445.513} C_VEL
LIN {X 0,Y 356.001,Z 974.302,A -85,B 0,C 180,E1 14442.142,E2 14442.142} C_VEL
LIN {X 0,Y 364.311,Z 960.436,A -85,B 0,C 180,E1 14439.536,E2 14439.536} C_VEL
LIN {X 0,Y 374.958,Z 942.021,A -85,B 0,C 180,E1 14436.615,E2 14436.615} C_VEL
LIN {X 0,Y 384.383,Z 924.622,A -85,B 0,C 180,E1 14434.32,E2 14434.32} C_VEL
LIN {X 0,Y 386.184,Z 921.228,A -85,B 0,C 180,E1 14433.911,E2 14433.911} C_VEL
LIN {X 0,Y 388.447,Z 915.839,A -85,B 0,C 180,E1 14433.157,E2 14433.157} C_VEL
LIN {X 0,Y 391.993,Z 901.783,A -85,B 0,C 180,E1 14430.884,E2 14430.884} C_VEL
LIN {X 0,Y 393.991,Z 896.745,A -85,B 0,C 180,E1 14430.312,E2 14430.312} C_VEL
LIN {X 0,Y 402.496,Z 878.55,A -85,B 0,C 180,E1 14428.726,E2 14428.726} C_VEL
LIN {X 0,Y 411.77,Z 856.912,A -85,B 0,C 180,E1 14427.132,E2 14427.132} C_VEL
LIN {X 0,Y 420.115,Z 834.679,A -85,B 0,C 180,E1 14425.785,E2 14425.785} C_VEL
LIN {X 0,Y 426.445,Z 815.805,A -85,B 0,C 180,E1 14424.816,E2 14424.816} C_VEL
LIN {X 0,Y 433.386,Z 792.355,A -85,B 0,C 180,E1 14423.813,E2 14423.813} C_VEL
LIN {X 0,Y 439.516,Z 766.911,A -85,B 0,C 180,E1 14422.958,E2 14422.958} C_VEL
LIN {X 0,Y 443.78,Z 745.419,A -85,B 0,C 180,E1 14422.395,E2 14422.395} C_VEL
LIN {X 0,Y 447.706,Z 719.579,A -85,B 0,C 180,E1 14421.86,E2 14421.86} C_VEL
LIN {X 0,Y 451.938,Z 671.916,A -85,B 0,C 180,E1 14421.094,E2 14421.094} C_VEL
LIN {X 0,Y 467.716,Z 483.144,A -85,B 0,C 180,E1 14418.171,E2 14418.171} C_VEL
LIN {X 0,Y 462.326,Z 473.967,A -85,B 0,C 180,E1 14415.749,E2 14415.749} C_VEL
LIN {X 0,Y 456.941,Z 465.262,A -85,B 0,C 180,E1 14412.897,E2 14412.897} C_VEL
LIN {X 0,Y 453.614,Z 460.228,A -85,B 0,C 180,E1 14410.799,E2 14410.799} C_VEL
LIN {X 0,Y 450.985,Z 456.048,A -85,B 0,C 180,E1 14408.8,E2 14408.8} C_VEL
LIN {X 0,Y 448.133,Z 451.498,A -85,B 0,C 180,E1 14406.02,E2 14406.02} C_VEL
LIN {X 0,Y 445.68,Z 447.679,A -85,B 0,C 180,E1 14402.186,E2 14402.186} C_VEL
LIN {X 0,Y 445.34,Z 446.526,A -85,B 0,C 180,E1 14401.029,E2 14401.029} C_VEL
LIN {X 0,Y 445.354,Z 446.559,A -85,B 0,C 180,E1 14396.009,E2 14396.009} C_VEL
LIN {X 0,Y 448.06,Z 451.515,A -85,B 0,C 180,E1 14391.142,E2 14391.142} C_VEL
LIN {X 0,Y 448.863,Z 452.808,A -85,B 0,C 180,E1 14390.253,E2 14390.253} C_VEL
LIN {X 0,Y 451.757,Z 457.263,A -85,B 0,C 180,E1 14387.667,E2 14387.667} C_VEL
LIN {X 0,Y 455.221,Z 462.644,A -85,B 0,C 180,E1 14385.239,E2 14385.239} C_VEL
LIN {X 0,Y 458.665,Z 468.203,A -85,B 0,C 180,E1 14383.211,E2 14383.211} C_VEL
LIN {X 0,Y 463.471,Z 476.057,A -85,B 0,C 180,E1 14380.792,E2 14380.792} C_VEL
LIN {X 0,Y 467.701,Z 484.234,A -85,B 0,C 180,E1 14378.88,E2 14378.88} C_VEL
LIN {X 0,Y 448.693,Z 711.405,A -85,B 0,C 180,E1 14375.352,E2 14375.352} C_VEL
LIN {X 0,Y 445.98,Z 733.944,A -85,B 0,C 180,E1 14374.946,E2 14374.946} C_VEL
LIN {X 0,Y 441.859,Z 758.378,A -85,B 0,C 180,E1 14374.402,E2 14374.402} C_VEL
LIN {X 0,Y 436.406,Z 782.811,A -85,B 0,C 180,E1 14373.692,E2 14373.692} C_VEL
LIN {X 0,Y 430.728,Z 804.05,A -85,B 0,C 180,E1 14372.919,E2 14372.919} C_VEL
LIN {X 0,Y 423.842,Z 826.447,A -85,B 0,C 180,E1 14371.921,E2 14371.921} C_VEL
LIN {X 0,Y 415.373,Z 850.129,A -85,B 0,C 180,E1 14370.622,E2 14370.622} C_VEL
LIN {X 0,Y 407.816,Z 868.989,A -85,B 0,C 180,E1 14369.382,E2 14369.382} C_VEL
LIN {X 0,Y 399.789,Z 887.289,A -85,B 0,C 180,E1 14367.978,E2 14367.978} C_VEL
LIN {X 0,Y 389.501,Z 908.837,A -85,B 0,C 180,E1 14366.014,E2 14366.014} C_VEL
LIN {X 0,Y 379.665,Z 927.601,A -85,B 0,C 180,E1 14363.951,E2 14363.951} C_VEL
LIN {X 0,Y 370.581,Z 943.976,A -85,B 0,C 180,E1 14361.838,E2 14361.838} C_VEL
LIN {X 0,Y 359.485,Z 962.953,A -85,B 0,C 180,E1 14358.918,E2 14358.918} C_VEL
LIN {X 0,Y 350.459,Z 977.63,A -85,B 0,C 180,E1 14356.206,E2 14356.206} C_VEL
LIN {X 0,Y 341.971,Z 991.154,A -85,B 0,C 180,E1 14353.276,E2 14353.276} C_VEL
LIN {X 0,Y 332.424,Z 1006.207,A -85,B 0,C 180,E1 14349.373,E2 14349.373} C_VEL
LIN {X 0,Y 325.051,Z 1017.87,A -85,B 0,C 180,E1 14345.699,E2 14345.699} C_VEL
LIN {X 0,Y 318.736,Z 1028.285,A -85,B 0,C 180,E1 14341.805,E2 14341.805} C_VEL
LIN {X 0,Y 312.807,Z 1038.735,A -85,B 0,C 180,E1 14336.994,E2 14336.994} C_VEL
LIN {X 0,Y 309.263,Z 1045.72,A -85,B 0,C 180,E1 14333.03,E2 14333.03} C_VEL
LIN {X 0,Y 306.654,Z 1051.766,A -85,B 0,C 180,E1 14328.833,E2 14328.833} C_VEL
LIN {X 0,Y 304.846,Z 1057.244,A -85,B 0,C 180,E1 14323.853,E2 14323.853} C_VEL
LIN {X 0,Y 304.141,Z 1060.465,A -85,B 0,C 180,E1 14319.652,E2 14319.652} C_VEL
LIN {X 0,Y 303.936,Z 1062.297,A -85,B 0,C 180,E1 14316.043,E2 14316.043} C_VEL
LIN {X 0,Y 303.912,Z 1063.229,A -85,B 0,C 180,E1 14312.451,E2 14312.451} C_VEL
LIN {X 0,Y 303.914,Z 1063.285,A -85,B 0,C 180,E1 14309.058,E2 14309.058} C_VEL
LIN {X 0,Y 303.91,Z 1062.53,A -85,B 0,C 180,E1 14305.66,E2 14305.66} C_VEL
LIN {X 0,Y 304.024,Z 1060.843,A -85,B 0,C 180,E1 14302.06,E2 14302.06} C_VEL
LIN {X 0,Y 304.394,Z 1058.074,A -85,B 0,C 180,E1 14298.249,E2 14298.249} C_VEL
LIN {X 0,Y 305.353,Z 1054.061,A -85,B 0,C 180,E1 14294.23,E2 14294.23} C_VEL
LIN {X 0,Y 307.593,Z 1047.437,A -85,B 0,C 180,E1 14289.248,E2 14289.248} C_VEL
LIN {X 0,Y 310.631,Z 1040.28,A -85,B 0,C 180,E1 14285.06,E2 14285.06} C_VEL
LIN {X 0,Y 314.599,Z 1032.154,A -85,B 0,C 180,E1 14281.112,E2 14281.112} C_VEL
LIN {X 0,Y 320.804,Z 1020.65,A -85,B 0,C 180,E1 14276.518,E2 14276.518} C_VEL
LIN {X 0,Y 327.288,Z 1009.23,A -85,B 0,C 180,E1 14272.778,E2 14272.778} C_VEL
LIN {X 0,Y 334.52,Z 996.86,A -85,B 0,C 180,E1 14269.337,E2 14269.337} C_VEL
LIN {X 0,Y 343.632,Z 981.21,A -85,B 0,C 180,E1 14265.706,E2 14265.706} C_VEL
LIN {X 0,Y 351.983,Z 966.617,A -85,B 0,C 180,E1 14262.87,E2 14262.87} C_VEL
LIN {X 0,Y 361.109,Z 950.291,A -85,B 0,C 180,E1 14260.162,E2 14260.162} C_VEL
LIN {X 0,Y 371.33,Z 930.922,A -85,B 0,C 180,E1 14257.485,E2 14257.485} C_VEL
LIN {X 0,Y 379.649,Z 914.201,A -85,B 0,C 180,E1 14255.53,E2 14255.53} C_VEL
LIN {X 0,Y 388.503,Z 895.281,A -85,B 0,C 180,E1 14253.635,E2 14253.635} C_VEL
LIN {X 0,Y 398.004,Z 872.996,A -85,B 0,C 180,E1 14251.772,E2 14251.772} C_VEL
LIN {X 0,Y 405.676,Z 853.13,A -85,B 0,C 180,E1 14250.384,E2 14250.384} C_VEL
LIN {X 0,Y 413.175,Z 831.667,A -85,B 0,C 180,E1 14249.118,E2 14249.118} C_VEL
LIN {X 0,Y 420.728,Z 806.609,A -85,B 0,C 180,E1 14247.917,E2 14247.917} C_VEL
LIN {X 0,Y 426.063,Z 786.047,A -85,B 0,C 180,E1 14247.117,E2 14247.117} C_VEL
LIN {X 0,Y 430.88,Z 764.141,A -85,B 0,C 180,E1 14246.416,E2 14246.416} C_VEL
LIN {X 0,Y 435.61,Z 736.652,A -85,B 0,C 180,E1 14245.748,E2 14245.748} C_VEL
LIN {X 0,Y 438.309,Z 714.013,A -85,B 0,C 180,E1 14245.32,E2 14245.32} C_VEL
LIN {X 0,Y 456.187,Z 487.347,A -85,B 0,C 180,E1 14241.735,E2 14241.735} C_VEL
LIN {X 0,Y 456.992,Z 477.024,A -85,B 0,C 180,E1 14241.567,E2 14241.567} C_VEL
LIN {X 0,Y 451.085,Z 465.952,A -85,B 0,C 180,E1 14239.252,E2 14239.252} C_VEL
LIN {X 0,Y 444.352,Z 455.079,A -85,B 0,C 180,E1 14236.269,E2 14236.269} C_VEL
LIN {X 0,Y 438.553,Z 446.17,A -85,B 0,C 180,E1 14233.179,E2 14233.179} C_VEL
LIN {X 0,Y 434.964,Z 440.919,A -85,B 0,C 180,E1 14230.865,E2 14230.865} C_VEL
LIN {X 0,Y 431.995,Z 436.461,A -85,B 0,C 180,E1 14228.519,E2 14228.519} C_VEL
LIN {X 0,Y 429.172,Z 432.053,A -85,B 0,C 180,E1 14225.548,E2 14225.548} C_VEL
LIN {X 0,Y 426.392,Z 428.292,A -85,B 0,C 180,E1 14219.463,E2 14219.463} C_VEL
LIN {X 0,Y 426.395,Z 428.322,A -85,B 0,C 180,E1 14217.312,E2 14217.312} C_VEL
LIN {X 0,Y 429.16,Z 432.014,A -85,B 0,C 180,E1 14211.289,E2 14211.289} C_VEL
LIN {X 0,Y 431.905,Z 436.344,A -85,B 0,C 180,E1 14208.38,E2 14208.38} C_VEL
LIN {X 0,Y 433.213,Z 438.406,A -85,B 0,C 180,E1 14207.266,E2 14207.266} C_VEL
LIN {X 0,Y 436.18,Z 442.689,A -85,B 0,C 180,E1 14205.123,E2 14205.123} C_VEL
LIN {X 0,Y 439.741,Z 448.146,A -85,B 0,C 180,E1 14202.943,E2 14202.943} C_VEL
LIN {X 0,Y 444.448,Z 455.158,A -85,B 0,C 180,E1 14200.508,E2 14200.508} C_VEL
LIN {X 0,Y 451.414,Z 466.512,A -85,B 0,C 180,E1 14197.434,E2 14197.434} C_VEL
LIN {X 0,Y 457.022,Z 475.989,A -85,B 0,C 180,E1 14195.286,E2 14195.286} C_VEL
LIN {X 0,Y 439.425,Z 700.436,A -85,B 0,C 180,E1 14191.748,E2 14191.748} C_VEL
LIN {X 0,Y 436.576,Z 727.315,A -85,B 0,C 180,E1 14191.265,E2 14191.265} C_VEL
LIN {X 0,Y 433.233,Z 749.005,A -85,B 0,C 180,E1 14190.773,E2 14190.773} C_VEL
LIN {X 0,Y 428.471,Z 773.398,A -85,B 0,C 180,E1 14190.068,E2 14190.068} C_VEL
LIN {X 0,Y 422.617,Z 797.052,A -85,B 0,C 180,E1 14189.186,E2 14189.186} C_VEL
LIN {X 0,Y 416.781,Z 817.404,A -85,B 0,C 180,E1 14188.262,E2 14188.262} C_VEL
LIN {X 0,Y 409.751,Z 839.115,A -85,B 0,C 180,E1 14187.08,E2 14187.08} C_VEL
LIN {X 0,Y 401.026,Z 862.562,A -85,B 0,C 180,E1 14185.529,E2 14185.529} C_VEL
LIN {X 0,Y 393.664,Z 880.474,A -85,B 0,C 180,E1 14184.119,E2 14184.119} C_VEL
LIN {X 0,Y 385.717,Z 898.341,A -85,B 0,C 180,E1 14182.489,E2 14182.489} C_VEL
LIN {X 0,Y 375.221,Z 920.1,A -85,B 0,C 180,E1 14180.126,E2 14180.126} C_VEL
LIN {X 0,Y 366.402,Z 937.04,A -85,B 0,C 180,E1 14177.925,E2 14177.925} C_VEL
LIN {X 0,Y 358.115,Z 952.247,A -85,B 0,C 180,E1 14175.624,E2 14175.624} C_VEL
LIN {X 0,Y 347.796,Z 970.39,A -85,B 0,C 180,E1 14172.365,E2 14172.365} C_VEL
LIN {X 0,Y 339.843,Z 983.903,A -85,B 0,C 180,E1 14169.458,E2 14169.458} C_VEL
LIN {X 0,Y 332.322,Z 996.622,A -85,B 0,C 180,E1 14166.258,E2 14166.258} C_VEL
LIN {X 0,Y 323.836,Z 1011.076,A -85,B 0,C 180,E1 14161.869,E2 14161.869} C_VEL
LIN {X 0,Y 318.069,Z 1021.214,A -85,B 0,C 180,E1 14158.134,E2 14158.134} C_VEL
LIN {X 0,Y 312.839,Z 1031.188,A -85,B 0,C 180,E1 14153.748,E2 14153.748} C_VEL
LIN {X 0,Y 308.829,Z 1039.58,A -85,B 0,C 180,E1 14149.087,E2 14149.087} C_VEL
LIN {X 0,Y 306.53,Z 1045.363,A -85,B 0,C 180,E1 14145.127,E2 14145.127} C_VEL
LIN {X 0,Y 305.024,Z 1050.205,A -85,B 0,C 180,E1 14140.96,E2 14140.96} C_VEL
LIN {X 0,Y 304.182,Z 1054.181,A -85,B 0,C 180,E1 14136.227,E2 14136.227} C_VEL
LIN {X 0,Y 303.947,Z 1056.282,A -85,B 0,C 180,E1 14132.262,E2 14132.262} C_VEL
LIN {X 0,Y 303.91,Z 1057.279,A -85,B 0,C 180,E1 14128.68,E2 14128.68} C_VEL
LIN {X 0,Y 303.912,Z 1057.396,A -85,B 0,C 180,E1 14125.093,E2 14125.093} C_VEL
LIN {X 0,Y 303.966,Z 1056.629,A -85,B 0,C 180,E1 14121.487,E2 14121.487} C_VEL
LIN {X 0,Y 304.187,Z 1054.969,A -85,B 0,C 180,E1 14117.856,E2 14117.856} C_VEL
LIN {X 0,Y 304.83,Z 1052.208,A -85,B 0,C 180,E1 14113.965,E2 14113.965} C_VEL
LIN {X 0,Y 306.314,Z 1047.842,A -85,B 0,C 180,E1 14109.529,E2 14109.529} C_VEL
LIN {X 0,Y 309.232,Z 1041.115,A -85,B 0,C 180,E1 14104.529,E2 14104.529} C_VEL
LIN {X 0,Y 312.771,Z 1034.28,A -85,B 0,C 180,E1 14100.507,E2 14100.507} C_VEL
LIN {X 0,Y 317.712,Z 1025.756,A -85,B 0,C 180,E1 14096.365,E2 14096.365} C_VEL
LIN {X 0,Y 324.567,Z 1014.585,A -85,B 0,C 180,E1 14091.966,E2 14091.966} C_VEL
LIN {X 0,Y 331.504,Z 1003.717,A -85,B 0,C 180,E1 14088.42,E2 14088.42} C_VEL
LIN {X 0,Y 340.329,Z 990.135,A -85,B 0,C 180,E1 14084.684,E2 14084.684} C_VEL
LIN {X 0,Y 349.923,Z 974.971,A -85,B 0,C 180,E1 14081.279,E2 14081.279} C_VEL
LIN {X 0,Y 358.496,Z 961.162,A -85,B 0,C 180,E1 14078.652,E2 14078.652} C_VEL
LIN {X 0,Y 369.064,Z 943.587,A -85,B 0,C 180,E1 14075.817,E2 14075.817} C_VEL
LIN {X 0,Y 379.44,Z 924.995,A -85,B 0,C 180,E1 14073.348,E2 14073.348} C_VEL
LIN {X 0,Y 388.111,Z 908.561,A -85,B 0,C 180,E1 14071.488,E2 14071.488} C_VEL
LIN {X 0,Y 393.991,Z 896.745,A -85,B 0,C 180,E1 14070.312,E2 14070.312} C_VEL
LIN {X 0,Y 396.278,Z 890.956,A -85,B 0,C 180,E1 14069.645,E2 14069.645} C_VEL
LIN {X 0,Y 399.895,Z 876.652,A -85,B 0,C 180,E1 14067.667,E2 14067.667} C_VEL
LIN {X 0,Y 402.108,Z 870.482,A -85,B 0,C 180,E1 14067.077,E2 14067.077} C_VEL
LIN {X 0,Y 410.624,Z 850.039,A -85,B 0,C 180,E1 14065.686,E2 14065.686} C_VEL
LIN {X 0,Y 418.197,Z 829.88,A -85,B 0,C 180,E1 14064.529,E2 14064.529} C_VEL
LIN {X 0,Y 426.555,Z 804.263,A -85,B 0,C 180,E1 14063.322,E2 14063.322} C_VEL
LIN {X 0,Y 432.223,Z 783.788,A -85,B 0,C 180,E1 14062.541,E2 14062.541} C_VEL
LIN {X 0,Y 437.219,Z 762.481,A -85,B 0,C 180,E1 14061.868,E2 14061.868} C_VEL
LIN {X 0,Y 442.241,Z 735.834,A -85,B 0,C 180,E1 14061.223,E2 14061.223} C_VEL
LIN {X 0,Y 445.39,Z 711.783,A -85,B 0,C 180,E1 14060.78,E2 14060.78} C_VEL
LIN {X 0,Y 464.623,Z 488.399,A -85,B 0,C 180,E1 14057.325,E2 14057.325} C_VEL
LIN {X 0,Y 460.082,Z 480.579,A -85,B 0,C 180,E1 14055.182,E2 14055.182} C_VEL
LIN {X 0,Y 455.315,Z 472.658,A -85,B 0,C 180,E1 14052.557,E2 14052.557} C_VEL
LIN {X 0,Y 452.175,Z 467.787,A -85,B 0,C 180,E1 14050.511,E2 14050.511} C_VEL
LIN {X 0,Y 449.695,Z 463.754,A -85,B 0,C 180,E1 14048.567,E2 14048.567} C_VEL
LIN {X 0,Y 446.924,Z 459.281,A -85,B 0,C 180,E1 14045.778,E2 14045.778} C_VEL
LIN {X 0,Y 444.609,Z 455.4,A -85,B 0,C 180,E1 14041.933,E2 14041.933} C_VEL
LIN {X 0,Y 444.325,Z 454.44,A -85,B 0,C 180,E1 14040.903,E2 14040.903} C_VEL
LIN {X 0,Y 444.423,Z 454.531,A -85,B 0,C 180,E1 14035.871,E2 14035.871} C_VEL
LIN {X 0,Y 446.639,Z 459.094,A -85,B 0,C 180,E1 14031.633,E2 14031.633} C_VEL
LIN {X 0,Y 447.48,Z 460.14,A -85,B 0,C 180,E1 14030.677,E2 14030.677} C_VEL
LIN {X 0,Y 450.532,Z 465.112,A -85,B 0,C 180,E1 14027.828,E2 14027.828} C_VEL
LIN {X 0,Y 453.845,Z 470.36,A -85,B 0,C 180,E1 14025.454,E2 14025.454} C_VEL
LIN {X 0,Y 458.246,Z 477.481,A -85,B 0,C 180,E1 14022.868,E2 14022.868} C_VEL
LIN {X 0,Y 462.387,Z 484.74,A -85,B 0,C 180,E1 14020.778,E2 14020.778} C_VEL
LIN {X 0,Y 464.593,Z 489.439,A -85,B 0,C 180,E1 14019.732,E2 14019.732} C_VEL
LIN {X 0,Y 445.292,Z 714.151,A -85,B 0,C 180,E1 14016.254,E2 14016.254} C_VEL
LIN {X 0,Y 442.378,Z 736.894,A -85,B 0,C 180,E1 14015.839,E2 14015.839} C_VEL
LIN {X 0,Y 437.215,Z 764.844,A -85,B 0,C 180,E1 14015.19,E2 14015.19} C_VEL
LIN {X 0,Y 432.485,Z 785.02,A -85,B 0,C 180,E1 14014.583,E2 14014.583} C_VEL
LIN {X 0,Y 426.732,Z 805.877,A -85,B 0,C 180,E1 14013.82,E2 14013.82} C_VEL
LIN {X 0,Y 419.035,Z 830.009,A -85,B 0,C 180,E1 14012.732,E2 14012.732} C_VEL
LIN {X 0,Y 410.759,Z 852.194,A -85,B 0,C 180,E1 14011.493,E2 14011.493} C_VEL
LIN {X 0,Y 403.026,Z 870.92,A -85,B 0,C 180,E1 14010.251,E2 14010.251} C_VEL
LIN {X 0,Y 393.245,Z 892.516,A -85,B 0,C 180,E1 14008.56,E2 14008.56} C_VEL
LIN {X 0,Y 383.065,Z 912.625,A -85,B 0,C 180,E1 14006.644,E2 14006.644} C_VEL
LIN {X 0,Y 373.979,Z 929.396,A -85,B 0,C 180,E1 14004.765,E2 14004.765} C_VEL
LIN {X 0,Y 363.025,Z 948.513,A -85,B 0,C 180,E1 14002.231,E2 14002.231} C_VEL
LIN {X 0,Y 352.501,Z 965.563,A -85,B 0,C 180,E1 13999.481,E2 13999.481} C_VEL
LIN {X 0,Y 343.755,Z 979.285,A -85,B 0,C 180,E1 13996.878,E2 13996.878} C_VEL
LIN {X 0,Y 333.992,Z 994.319,A -85,B 0,C 180,E1 13993.516,E2 13993.516} C_VEL
LIN {X 0,Y 324.903,Z 1007.899,A -85,B 0,C 180,E1 13989.801,E2 13989.801} C_VEL
LIN {X 0,Y 317.762,Z 1018.761,A -85,B 0,C 180,E1 13986.268,E2 13986.268} C_VEL
LIN {X 0,Y 310.472,Z 1030.311,A -85,B 0,C 180,E1 13981.763,E2 13981.763} C_VEL
LIN {X 0,Y 305.031,Z 1039.429,A -85,B 0,C 180,E1 13977.317,E2 13977.317} C_VEL
LIN {X 0,Y 301.33,Z 1046.396,A -85,B 0,C 180,E1 13973.196,E2 13973.196} C_VEL
LIN {X 0,Y 298.32,Z 1053.196,A -85,B 0,C 180,E1 13968.162,E2 13968.162} C_VEL
LIN {X 0,Y 296.746,Z 1057.839,A -85,B 0,C 180,E1 13963.444,E2 13963.444} C_VEL
LIN {X 0,Y 296.127,Z 1060.637,A -85,B 0,C 180,E1 13959.523,E2 13959.523} C_VEL
LIN {X 0,Y 295.929,Z 1062.369,A -85,B 0,C 180,E1 13955.818,E2 13955.818} C_VEL
LIN {X 0,Y 295.908,Z 1063.202,A -85,B 0,C 180,E1 13952.13,E2 13952.13} C_VEL
LIN {X 0,Y 295.911,Z 1063.158,A -85,B 0,C 180,E1 13948.645,E2 13948.645} C_VEL
LIN {X 0,Y 295.912,Z 1062.302,A -85,B 0,C 180,E1 13945.154,E2 13945.154} C_VEL
LIN {X 0,Y 296.051,Z 1060.514,A -85,B 0,C 180,E1 13941.454,E2 13941.454} C_VEL
LIN {X 0,Y 296.55,Z 1057.48,A -85,B 0,C 180,E1 13937.34,E2 13937.34} C_VEL
LIN {X 0,Y 298.073,Z 1052.113,A -85,B 0,C 180,E1 13932.226,E2 13932.226} C_VEL
LIN {X 0,Y 300.391,Z 1046.07,A -85,B 0,C 180,E1 13927.906,E2 13927.906} C_VEL
LIN {X 0,Y 303.656,Z 1039.057,A -85,B 0,C 180,E1 13923.817,E2 13923.817} C_VEL
LIN {X 0,Y 309.001,Z 1029.021,A -85,B 0,C 180,E1 13919.036,E2 13919.036} C_VEL
LIN {X 0,Y 315.08,Z 1018.382,A -85,B 0,C 180,E1 13914.943,E2 13914.943} C_VEL
LIN {X 0,Y 321.38,Z 1007.875,A -85,B 0,C 180,E1 13911.52,E2 13911.52} C_VEL
LIN {X 0,Y 329.867,Z 994,A -85,B 0,C 180,E1 13907.699,E2 13907.699} C_VEL
LIN {X 0,Y 338.63,Z 979.416,A -85,B 0,C 180,E1 13904.393,E2 13904.393} C_VEL
LIN {X 0,Y 346.876,Z 965.514,A -85,B 0,C 180,E1 13901.705,E2 13901.705} C_VEL
LIN {X 0,Y 357.178,Z 947.625,A -85,B 0,C 180,E1 13898.773,E2 13898.773} C_VEL
LIN {X 0,Y 366.819,Z 929.71,A -85,B 0,C 180,E1 13896.343,E2 13896.343} C_VEL
LIN {X 0,Y 375.213,Z 913.263,A -85,B 0,C 180,E1 13894.435,E2 13894.435} C_VEL
LIN {X 0,Y 384.973,Z 892.91,A -85,B 0,C 180,E1 13892.423,E2 13892.423} C_VEL
LIN {X 0,Y 394.143,Z 871.615,A -85,B 0,C 180,E1 13890.684,E2 13890.684} C_VEL
LIN {X 0,Y 401.616,Z 852.634,A -85,B 0,C 180,E1 13889.371,E2 13889.371} C_VEL
LIN {X 0,Y 409.709,Z 829.9,A -85,B 0,C 180,E1 13888.047,E2 13888.047} C_VEL
LIN {X 0,Y 417.106,Z 805.529,A -85,B 0,C 180,E1 13886.906,E2 13886.906} C_VEL
LIN {X 0,Y 422.408,Z 785.429,A -85,B 0,C 180,E1 13886.137,E2 13886.137} C_VEL
LIN {X 0,Y 427.36,Z 763.276,A -85,B 0,C 180,E1 13885.44,E2 13885.44} C_VEL
LIN {X 0,Y 432.06,Z 736.198,A -85,B 0,C 180,E1 13884.793,E2 13884.793} C_VEL
LIN {X 0,Y 434.775,Z 713.763,A -85,B 0,C 180,E1 13884.372,E2 13884.372} C_VEL
LIN {X 0,Y 453.078,Z 487.404,A -85,B 0,C 180,E1 13880.803,E2 13880.803} C_VEL
LIN {X 0,Y 453.508,Z 481.637,A -85,B 0,C 180,E1 13880.7,E2 13880.7} C_VEL
LIN {X 0,Y 448.664,Z 472.477,A -85,B 0,C 180,E1 13878.719,E2 13878.719} C_VEL
LIN {X 0,Y 442.447,Z 462.259,A -85,B 0,C 180,E1 13875.87,E2 13875.87} C_VEL
LIN {X 0,Y 437.021,Z 453.717,A -85,B 0,C 180,E1 13872.89,E2 13872.89} C_VEL
LIN {X 0,Y 433.519,Z 448.492,A -85,B 0,C 180,E1 13870.566,E2 13870.566} C_VEL
LIN {X 0,Y 430.711,Z 444.181,A -85,B 0,C 180,E1 13868.275,E2 13868.275} C_VEL
LIN {X 0,Y 427.989,Z 439.735,A -85,B 0,C 180,E1 13865.295,E2 13865.295} C_VEL
LIN {X 0,Y 425.378,Z 436.109,A -85,B 0,C 180,E1 13858.922,E2 13858.922} C_VEL
LIN {X 0,Y 425.524,Z 436.701,A -85,B 0,C 180,E1 13856.497,E2 13856.497} C_VEL
LIN {X 0,Y 428.028,Z 439.831,A -85,B 0,C 180,E1 13851.469,E2 13851.469} C_VEL
LIN {X 0,Y 430.783,Z 444.23,A -85,B 0,C 180,E1 13848.485,E2 13848.485} C_VEL
LIN {X 0,Y 434.717,Z 450.24,A -85,B 0,C 180,E1 13845.412,E2 13845.412} C_VEL
LIN {X 0,Y 438.305,Z 455.879,A -85,B 0,C 180,E1 13843.159,E2 13843.159} C_VEL
LIN {X 0,Y 442.853,Z 462.847,A -85,B 0,C 180,E1 13840.753,E2 13840.753} C_VEL
LIN {X 0,Y 450.265,Z 475.069,A -85,B 0,C 180,E1 13837.442,E2 13837.442} C_VEL
LIN {X 0,Y 453.54,Z 481.047,A -85,B 0,C 180,E1 13836.135,E2 13836.135} C_VEL
LIN {X 0,Y 435.029,Z 709.635,A -85,B 0,C 180,E1 13832.536,E2 13832.536} C_VEL
LIN {X 0,Y 432.358,Z 731.861,A -85,B 0,C 180,E1 13832.12,E2 13832.12} C_VEL
LIN {X 0,Y 427.887,Z 758.249,A -85,B 0,C 180,E1 13831.488,E2 13831.488} C_VEL
LIN {X 0,Y 422.851,Z 781.136,A -85,B 0,C 180,E1 13830.756,E2 13830.756} C_VEL
LIN {X 0,Y 417.887,Z 800.257,A -85,B 0,C 180,E1 13830.016,E2 13830.016} C_VEL
LIN {X 0,Y 411.366,Z 822.122,A -85,B 0,C 180,E1 13829.001,E2 13829.001} C_VEL
LIN {X 0,Y 403.076,Z 846.086,A -85,B 0,C 180,E1 13827.635,E2 13827.635} C_VEL
LIN {X 0,Y 395.441,Z 865.664,A -85,B 0,C 180,E1 13826.293,E2 13826.293} C_VEL
LIN {X 0,Y 387.089,Z 885.251,A -85,B 0,C 180,E1 13824.712,E2 13824.712} C_VEL
LIN {X 0,Y 376.563,Z 907.551,A -85,B 0,C 180,E1 13822.55,E2 13822.55} C_VEL
LIN {X 0,Y 368.077,Z 924.199,A -85,B 0,C 180,E1 13820.628,E2 13820.628} C_VEL
LIN {X 0,Y 359.093,Z 940.86,A -85,B 0,C 180,E1 13818.386,E2 13818.386} C_VEL
LIN {X 0,Y 348.385,Z 959.548,A -85,B 0,C 180,E1 13815.379,E2 13815.379} C_VEL
LIN {X 0,Y 339.749,Z 973.993,A -85,B 0,C 180,E1 13812.601,E2 13812.601} C_VEL
LIN {X 0,Y 331.022,Z 988.36,A -85,B 0,C 180,E1 13809.35,E2 13809.35} C_VEL
LIN {X 0,Y 322.256,Z 1002.53,A -85,B 0,C 180,E1 13805.466,E2 13805.466} C_VEL
LIN {X 0,Y 315.662,Z 1013.311,A -85,B 0,C 180,E1 13801.937,E2 13801.937} C_VEL
LIN {X 0,Y 309.131,Z 1024.568,A -85,B 0,C 180,E1 13797.551,E2 13797.551} C_VEL
LIN {X 0,Y 303.893,Z 1034.101,A -85,B 0,C 180,E1 13792.886,E2 13792.886} C_VEL
LIN {X 0,Y 300.606,Z 1040.928,A -85,B 0,C 180,E1 13788.823,E2 13788.823} C_VEL
LIN {X 0,Y 298.028,Z 1047.483,A -85,B 0,C 180,E1 13783.979,E2 13783.979} C_VEL
LIN {X 0,Y 296.64,Z 1052.071,A -85,B 0,C 180,E1 13779.311,E2 13779.311} C_VEL
LIN {X 0,Y 296.116,Z 1054.848,A -85,B 0,C 180,E1 13775.425,E2 13775.425} C_VEL
LIN {X 0,Y 295.935,Z 1056.579,A -85,B 0,C 180,E1 13771.742,E2 13771.742} C_VEL
LIN {X 0,Y 295.908,Z 1057.385,A -85,B 0,C 180,E1 13768.451,E2 13768.451} C_VEL
LIN {X 0,Y 295.916,Z 1057.446,A -85,B 0,C 180,E1 13764.765,E2 13764.765} C_VEL
LIN {X 0,Y 295.971,Z 1056.691,A -85,B 0,C 180,E1 13761.256,E2 13761.256} C_VEL
LIN {X 0,Y 296.222,Z 1055.02,A -85,B 0,C 180,E1 13757.524,E2 13757.524} C_VEL
LIN {X 0,Y 296.926,Z 1052.282,A -85,B 0,C 180,E1 13753.569,E2 13753.569} C_VEL
LIN {X 0,Y 298.54,Z 1047.9,A -85,B 0,C 180,E1 13749,E2 13749} C_VEL
LIN {X 0,Y 301.698,Z 1041.12,A -85,B 0,C 180,E1 13743.846,E2 13743.846} C_VEL
LIN {X 0,Y 305.482,Z 1034.273,A -85,B 0,C 180,E1 13739.731,E2 13739.731} C_VEL
LIN {X 0,Y 310.99,Z 1025.331,A -85,B 0,C 180,E1 13735.313,E2 13735.313} C_VEL
LIN {X 0,Y 318.298,Z 1014.021,A -85,B 0,C 180,E1 13730.846,E2 13730.846} C_VEL
LIN {X 0,Y 325.212,Z 1003.675,A -85,B 0,C 180,E1 13727.437,E2 13727.437} C_VEL
LIN {X 0,Y 334.447,Z 990.059,A -85,B 0,C 180,E1 13723.656,E2 13723.656} C_VEL
LIN {X 0,Y 344.429,Z 974.863,A -85,B 0,C 180,E1 13720.227,E2 13720.227} C_VEL
LIN {X 0,Y 353.315,Z 961.037,A -85,B 0,C 180,E1 13717.589,E2 13717.589} C_VEL
LIN {X 0,Y 364.296,Z 943.305,A -85,B 0,C 180,E1 13714.733,E2 13714.733} C_VEL
LIN {X 0,Y 374.609,Z 925.368,A -85,B 0,C 180,E1 13712.351,E2 13712.351} C_VEL
LIN {X 0,Y 383.548,Z 908.893,A -85,B 0,C 180,E1 13710.487,E2 13710.487} C_VEL
LIN {X 0,Y 394.104,Z 888.035,A -85,B 0,C 180,E1 13708.488,E2 13708.488} C_VEL
LIN {X 0,Y 402.108,Z 870.482,A -85,B 0,C 180,E1 13707.077,E2 13707.077} C_VEL
LIN {X 0,Y 404.369,Z 864.211,A -85,B 0,C 180,E1 13706.508,E2 13706.508} C_VEL
LIN {X 0,Y 408.197,Z 848.059,A -85,B 0,C 180,E1 13704.642,E2 13704.642} C_VEL
LIN {X 0,Y 410.069,Z 842.493,A -85,B 0,C 180,E1 13704.208,E2 13704.208} C_VEL
LIN {X 0,Y 418.24,Z 819.731,A -85,B 0,C 180,E1 13703.013,E2 13703.013} C_VEL
LIN {X 0,Y 424.86,Z 798.712,A -85,B 0,C 180,E1 13702.101,E2 13702.101} C_VEL
LIN {X 0,Y 431.308,Z 774.963,A -85,B 0,C 180,E1 13701.261,E2 13701.261} C_VEL
LIN {X 0,Y 436.711,Z 749.773,A -85,B 0,C 180,E1 13700.573,E2 13700.573} C_VEL
LIN {X 0,Y 440.308,Z 728.388,A -85,B 0,C 180,E1 13700.115,E2 13700.115} C_VEL
LIN {X 0,Y 443.405,Z 702.309,A -85,B 0,C 180,E1 13699.661,E2 13699.661} C_VEL
LIN {X 0,Y 461.607,Z 493.54,A -85,B 0,C 180,E1 13696.453,E2 13696.453} C_VEL
LIN {X 0,Y 456.21,Z 484.216,A -85,B 0,C 180,E1 13693.692,E2 13693.692} C_VEL
LIN {X 0,Y 452.539,Z 478.227,A -85,B 0,C 180,E1 13691.47,E2 13691.47} C_VEL
LIN {X 0,Y 450.241,Z 474.575,A -85,B 0,C 180,E1 13689.846,E2 13689.846} C_VEL
LIN {X 0,Y 448.413,Z 471.458,A -85,B 0,C 180,E1 13688.334,E2 13688.334} C_VEL
LIN {X 0,Y 445.835,Z 467.16,A -85,B 0,C 180,E1 13685.663,E2 13685.663} C_VEL
LIN {X 0,Y 443.547,Z 463.118,A -85,B 0,C 180,E1 13681.679,E2 13681.679} C_VEL
LIN {X 0,Y 443.313,Z 462.356,A -85,B 0,C 180,E1 13680.775,E2 13680.775} C_VEL
LIN {X 0,Y 443.407,Z 462.447,A -85,B 0,C 180,E1 13675.991,E2 13675.991} C_VEL
LIN {X 0,Y 445.561,Z 466.976,A -85,B 0,C 180,E1 13671.742,E2 13671.742} C_VEL
LIN {X 0,Y 446.382,Z 468.077,A -85,B 0,C 180,E1 13670.784,E2 13670.784} C_VEL
LIN {X 0,Y 449.238,Z 472.811,A -85,B 0,C 180,E1 13668.054,E2 13668.054} C_VEL
LIN {X 0,Y 452.476,Z 478.073,A -85,B 0,C 180,E1 13665.67,E2 13665.67} C_VEL
LIN {X 0,Y 456.628,Z 484.956,A -85,B 0,C 180,E1 13663.166,E2 13663.166} C_VEL
LIN {X 0,Y 460.556,Z 492.007,A -85,B 0,C 180,E1 13661.126,E2 13661.126} C_VEL
LIN {X 0,Y 461.604,Z 494.464,A -85,B 0,C 180,E1 13660.597,E2 13660.597} C_VEL
LIN {X 0,Y 442.104,Z 715.948,A -85,B 0,C 180,E1 13657.185,E2 13657.185} C_VEL
LIN {X 0,Y 438.551,Z 742.037,A -85,B 0,C 180,E1 13656.704,E2 13656.704} C_VEL
LIN {X 0,Y 433.492,Z 767.363,A -85,B 0,C 180,E1 13656.095,E2 13656.095} C_VEL
LIN {X 0,Y 428.605,Z 787.49,A -85,B 0,C 180,E1 13655.481,E2 13655.481} C_VEL
LIN {X 0,Y 421.769,Z 811.402,A -85,B 0,C 180,E1 13654.587,E2 13654.587} C_VEL
LIN {X 0,Y 413.543,Z 835.342,A -85,B 0,C 180,E1 13653.458,E2 13653.458} C_VEL
LIN {X 0,Y 405.879,Z 855.154,A -85,B 0,C 180,E1 13652.329,E2 13652.329} C_VEL
LIN {X 0,Y 396.288,Z 877.49,A -85,B 0,C 180,E1 13650.809,E2 13650.809} C_VEL
LIN {X 0,Y 386.292,Z 898.083,A -85,B 0,C 180,E1 13649.099,E2 13649.099} C_VEL
LIN {X 0,Y 377.324,Z 915.206,A -85,B 0,C 180,E1 13647.424,E2 13647.424} C_VEL
LIN {X 0,Y 366.521,Z 934.503,A -85,B 0,C 180,E1 13645.199,E2 13645.199} C_VEL
LIN {X 0,Y 355.684,Z 952.302,A -85,B 0,C 180,E1 13642.708,E2 13642.708} C_VEL
LIN {X 0,Y 346.638,Z 966.492,A -85,B 0,C 180,E1 13640.369,E2 13640.369} C_VEL
LIN {X 0,Y 337.165,Z 980.842,A -85,B 0,C 180,E1 13637.598,E2 13637.598} C_VEL
LIN {X 0,Y 326.193,Z 996.916,A -85,B 0,C 180,E1 13633.849,E2 13633.849} C_VEL
LIN {X 0,Y 317.741,Z 1009.101,A -85,B 0,C 180,E1 13630.399,E2 13630.399} C_VEL
LIN {X 0,Y 309.95,Z 1020.512,A -85,B 0,C 180,E1 13626.556,E2 13626.556} C_VEL
LIN {X 0,Y 302.263,Z 1032.047,A -85,B 0,C 180,E1 13621.771,E2 13621.771} C_VEL
LIN {X 0,Y 297.264,Z 1040.124,A -85,B 0,C 180,E1 13617.657,E2 13617.657} C_VEL
LIN {X 0,Y 293.042,Z 1047.807,A -85,B 0,C 180,E1 13612.887,E2 13612.887} C_VEL
LIN {X 0,Y 290.168,Z 1053.986,A -85,B 0,C 180,E1 13607.86,E2 13607.86} C_VEL
LIN {X 0,Y 288.779,Z 1057.95,A -85,B 0,C 180,E1 13603.618,E2 13603.618} C_VEL
LIN {X 0,Y 288.132,Z 1060.694,A -85,B 0,C 180,E1 13599.589,E2 13599.589} C_VEL
LIN {X 0,Y 287.928,Z 1062.372,A -85,B 0,C 180,E1 13595.78,E2 13595.78} C_VEL
LIN {X 0,Y 287.906,Z 1063.151,A -85,B 0,C 180,E1 13591.99,E2 13591.99} C_VEL
LIN {X 0,Y 287.907,Z 1063.03,A -85,B 0,C 180,E1 13588.209,E2 13588.209} C_VEL
LIN {X 0,Y 287.928,Z 1061.936,A -85,B 0,C 180,E1 13584.22,E2 13584.22} C_VEL
LIN {X 0,Y 288.204,Z 1059.474,A -85,B 0,C 180,E1 13579.607,E2 13579.607} C_VEL
LIN {X 0,Y 289.172,Z 1055.262,A -85,B 0,C 180,E1 13574.736,E2 13574.736} C_VEL
LIN {X 0,Y 290.831,Z 1050.438,A -85,B 0,C 180,E1 13570.519,E2 13570.519} C_VEL
LIN {X 0,Y 293.633,Z 1044.087,A -85,B 0,C 180,E1 13566.095,E2 13566.095} C_VEL
LIN {X 0,Y 298.501,Z 1034.709,A -85,B 0,C 180,E1 13560.942,E2 13560.942} C_VEL
LIN {X 0,Y 303.495,Z 1026.062,A -85,B 0,C 180,E1 13557.071,E2 13557.071} C_VEL
LIN {X 0,Y 309.841,Z 1015.701,A -85,B 0,C 180,E1 13553.161,E2 13553.161} C_VEL
LIN {X 0,Y 318.735,Z 1001.596,A -85,B 0,C 180,E1 13548.793,E2 13548.793} C_VEL
LIN {X 0,Y 326.8,Z 988.839,A -85,B 0,C 180,E1 13545.521,E2 13545.521} C_VEL
LIN {X 0,Y 335.787,Z 974.502,A -85,B 0,C 180,E1 13542.398,E2 13542.398} C_VEL
LIN {X 0,Y 346.448,Z 956.79,A -85,B 0,C 180,E1 13539.202,E2 13539.202} C_VEL
LIN {X 0,Y 355.154,Z 941.699,A -85,B 0,C 180,E1 13536.912,E2 13536.912} C_VEL
LIN {X 0,Y 364.385,Z 924.914,A -85,B 0,C 180,E1 13534.731,E2 13534.731} C_VEL
LIN {X 0,Y 375.595,Z 902.914,A -85,B 0,C 180,E1 13532.35,E2 13532.35} C_VEL
LIN {X 0,Y 383.92,Z 885.148,A -85,B 0,C 180,E1 13530.745,E2 13530.745} C_VEL
LIN {X 0,Y 392.085,Z 866.292,A -85,B 0,C 180,E1 13529.29,E2 13529.29} C_VEL
LIN {X 0,Y 401.549,Z 841.882,A -85,B 0,C 180,E1 13527.722,E2 13527.722} C_VEL
LIN {X 0,Y 408.608,Z 821.035,A -85,B 0,C 180,E1 13526.622,E2 13526.622} C_VEL
LIN {X 0,Y 414.96,Z 799.747,A -85,B 0,C 180,E1 13525.686,E2 13525.686} C_VEL
LIN {X 0,Y 421.819,Z 772.237,A -85,B 0,C 180,E1 13524.727,E2 13524.727} C_VEL
LIN {X 0,Y 426.263,Z 750.121,A -85,B 0,C 180,E1 13524.139,E2 13524.139} C_VEL
LIN {X 0,Y 430.125,Z 725.243,A -85,B 0,C 180,E1 13523.614,E2 13523.614} C_VEL
LIN {X 0,Y 433.668,Z 686.761,A -85,B 0,C 180,E1 13522.976,E2 13522.976} C_VEL
LIN {X 0,Y 450.153,Z 486.402,A -85,B 0,C 180,E1 13519.834,E2 13519.834} C_VEL
LIN {X 0,Y 446.354,Z 479.113,A -85,B 0,C 180,E1 13518.21,E2 13518.21} C_VEL
LIN {X 0,Y 440.564,Z 469.435,A -85,B 0,C 180,E1 13515.467,E2 13515.467} C_VEL
LIN {X 0,Y 435.395,Z 461.125,A -85,B 0,C 180,E1 13512.534,E2 13512.534} C_VEL
LIN {X 0,Y 432.174,Z 456.177,A -85,B 0,C 180,E1 13510.329,E2 13510.329} C_VEL
LIN {X 0,Y 429.435,Z 451.9,A -85,B 0,C 180,E1 13508.031,E2 13508.031} C_VEL
LIN {X 0,Y 426.655,Z 447.33,A -85,B 0,C 180,E1 13504.84,E2 13504.84} C_VEL
LIN {X 0,Y 424.396,Z 443.997,A -85,B 0,C 180,E1 13498.65,E2 13498.65} C_VEL
LIN {X 0,Y 424.664,Z 444.947,A -85,B 0,C 180,E1 13495.949,E2 13495.949} C_VEL
LIN {X 0,Y 426.944,Z 447.768,A -85,B 0,C 180,E1 13491.583,E2 13491.583} C_VEL
LIN {X 0,Y 429.814,Z 452.274,A -85,B 0,C 180,E1 13488.459,E2 13488.459} C_VEL
LIN {X 0,Y 433.445,Z 458.124,A -85,B 0,C 180,E1 13485.573,E2 13485.573} C_VEL
LIN {X 0,Y 436.875,Z 463.608,A -85,B 0,C 180,E1 13483.376,E2 13483.376} C_VEL
LIN {X 0,Y 441.159,Z 470.338,A -85,B 0,C 180,E1 13481.054,E2 13481.054} C_VEL
LIN {X 0,Y 448.287,Z 482.363,A -85,B 0,C 180,E1 13477.786,E2 13477.786} C_VEL
LIN {X 0,Y 450.162,Z 485.948,A -85,B 0,C 180,E1 13477.003,E2 13477.003} C_VEL
LIN {X 0,Y 431.398,Z 711.694,A -85,B 0,C 180,E1 13473.46,E2 13473.46} C_VEL
LIN {X 0,Y 428.32,Z 735.845,A -85,B 0,C 180,E1 13473.002,E2 13473.002} C_VEL
LIN {X 0,Y 423.421,Z 762.454,A -85,B 0,C 180,E1 13472.336,E2 13472.336} C_VEL
LIN {X 0,Y 418.467,Z 784.083,A -85,B 0,C 180,E1 13471.629,E2 13471.629} C_VEL
LIN {X 0,Y 412.538,Z 806,A -85,B 0,C 180,E1 13470.756,E2 13470.756} C_VEL
LIN {X 0,Y 404.749,Z 830.259,A -85,B 0,C 180,E1 13469.56,E2 13469.56} C_VEL
LIN {X 0,Y 397.468,Z 850.136,A -85,B 0,C 180,E1 13468.38,E2 13468.38} C_VEL
LIN {X 0,Y 389.036,Z 870.928,A -85,B 0,C 180,E1 13466.916,E2 13466.916} C_VEL
LIN {X 0,Y 378.932,Z 893.184,A -85,B 0,C 180,E1 13465.016,E2 13465.016} C_VEL
LIN {X 0,Y 370.158,Z 910.899,A -85,B 0,C 180,E1 13463.217,E2 13463.217} C_VEL
LIN {X 0,Y 360.296,Z 929.552,A -85,B 0,C 180,E1 13460.991,E2 13460.991} C_VEL
LIN {X 0,Y 349.583,Z 948.277,A -85,B 0,C 180,E1 13458.289,E2 13458.289} C_VEL
LIN {X 0,Y 340.649,Z 963.166,A -85,B 0,C 180,E1 13455.741,E2 13455.741} C_VEL
LIN {X 0,Y 330.53,Z 979.558,A -85,B 0,C 180,E1 13452.423,E2 13452.423} C_VEL
LIN {X 0,Y 321.431,Z 993.682,A -85,B 0,C 180,E1 13448.93,E2 13448.93} C_VEL
LIN {X 0,Y 314.152,Z 1005.01,A -85,B 0,C 180,E1 13445.623,E2 13445.623} C_VEL
LIN {X 0,Y 306.588,Z 1017.064,A -85,B 0,C 180,E1 13441.454,E2 13441.454} C_VEL
LIN {X 0,Y 300.163,Z 1027.553,A -85,B 0,C 180,E1 13436.938,E2 13436.938} C_VEL
LIN {X 0,Y 295.79,Z 1035.379,A -85,B 0,C 180,E1 13432.876,E2 13432.876} C_VEL
LIN {X 0,Y 292.005,Z 1043.138,A -85,B 0,C 180,E1 13427.949,E2 13427.949} C_VEL
LIN {X 0,Y 289.711,Z 1048.833,A -85,B 0,C 180,E1 13423.167,E2 13423.167} C_VEL
LIN {X 0,Y 288.578,Z 1052.66,A -85,B 0,C 180,E1 13418.97,E2 13418.97} C_VEL
LIN {X 0,Y 288.085,Z 1055.29,A -85,B 0,C 180,E1 13414.978,E2 13414.978} C_VEL
LIN {X 0,Y 287.942,Z 1057.01,A -85,B 0,C 180,E1 13410.796,E2 13410.796} C_VEL
LIN {X 0,Y 287.908,Z 1057.697,A -85,B 0,C 180,E1 13406.216,E2 13406.216} C_VEL
LIN {X 0,Y 287.96,Z 1056.996,A -85,B 0,C 180,E1 13401.737,E2 13401.737} C_VEL
LIN {X 0,Y 288.218,Z 1055.297,A -85,B 0,C 180,E1 13397.579,E2 13397.579} C_VEL
LIN {X 0,Y 288.955,Z 1052.583,A -85,B 0,C 180,E1 13393.441,E2 13393.441} C_VEL
LIN {X 0,Y 290.51,Z 1048.547,A -85,B 0,C 180,E1 13389.026,E2 13389.026} C_VEL
LIN {X 0,Y 293.886,Z 1041.732,A -85,B 0,C 180,E1 13383.532,E2 13383.532} C_VEL
LIN {X 0,Y 297.901,Z 1034.83,A -85,B 0,C 180,E1 13379.233,E2 13379.233} C_VEL
LIN {X 0,Y 303.241,Z 1026.53,A -85,B 0,C 180,E1 13374.989,E2 13374.989} C_VEL
LIN {X 0,Y 311.234,Z 1014.795,A -85,B 0,C 180,E1 13370.16,E2 13370.16} C_VEL
LIN {X 0,Y 318.63,Z 1004.192,A -85,B 0,C 180,E1 13366.588,E2 13366.588} C_VEL
LIN {X 0,Y 327.279,Z 991.901,A -85,B 0,C 180,E1 13363.099,E2 13363.099} C_VEL
LIN {X 0,Y 338.018,Z 976.307,A -85,B 0,C 180,E1 13359.461,E2 13359.461} C_VEL
LIN {X 0,Y 347.137,Z 962.616,A -85,B 0,C 180,E1 13356.799,E2 13356.799} C_VEL
LIN {X 0,Y 356.63,Z 947.81,A -85,B 0,C 180,E1 13354.341,E2 13354.341} C_VEL
LIN {X 0,Y 368.893,Z 927.504,A -85,B 0,C 180,E1 13351.543,E2 13351.543} C_VEL
LIN {X 0,Y 378.362,Z 910.594,A -85,B 0,C 180,E1 13349.607,E2 13349.607} C_VEL
LIN {X 0,Y 387.49,Z 893.127,A -85,B 0,C 180,E1 13347.897,E2 13347.897} C_VEL
LIN {X 0,Y 398.637,Z 869.692,A -85,B 0,C 180,E1 13345.987,E2 13345.987} C_VEL
LIN {X 0,Y 407.062,Z 849.858,A -85,B 0,C 180,E1 13344.653,E2 13344.653} C_VEL
LIN {X 0,Y 410.069,Z 842.493,A -85,B 0,C 180,E1 13344.208,E2 13344.208} C_VEL
LIN {X 0,Y 412.185,Z 835.934,A -85,B 0,C 180,E1 13343.71,E2 13343.71} C_VEL
LIN {X 0,Y 415.604,Z 818.767,A -85,B 0,C 180,E1 13342.049,E2 13342.049} C_VEL
LIN {X 0,Y 417.285,Z 812.909,A -85,B 0,C 180,E1 13341.686,E2 13341.686} C_VEL
LIN {X 0,Y 424.904,Z 787.665,A -85,B 0,C 180,E1 13340.689,E2 13340.689} C_VEL
LIN {X 0,Y 430.425,Z 765.446,A -85,B 0,C 180,E1 13339.986,E2 13339.986} C_VEL
LIN {X 0,Y 435.118,Z 742.57,A -85,B 0,C 180,E1 13339.422,E2 13339.422} C_VEL
LIN {X 0,Y 439.224,Z 714.741,A -85,B 0,C 180,E1 13338.893,E2 13338.893} C_VEL
LIN {X 0,Y 450.922,Z 585.121,A -85,B 0,C 180,E1 13336.894,E2 13336.894} C_VEL
LIN {X 0,Y 458.716,Z 498.924,A -85,B 0,C 180,E1 13335.588,E2 13335.588} C_VEL
LIN {X 0,Y 453.603,Z 490.009,A -85,B 0,C 180,E1 13332.799,E2 13332.799} C_VEL
LIN {X 0,Y 449.759,Z 483.519,A -85,B 0,C 180,E1 13330.245,E2 13330.245} C_VEL
LIN {X 0,Y 447.139,Z 479.161,A -85,B 0,C 180,E1 13328.099,E2 13328.099} C_VEL
LIN {X 0,Y 444.748,Z 475.038,A -85,B 0,C 180,E1 13325.548,E2 13325.548} C_VEL
LIN {X 0,Y 442.526,Z 470.996,A -85,B 0,C 180,E1 13321.554,E2 13321.554} C_VEL
LIN {X 0,Y 442.302,Z 470.273,A -85,B 0,C 180,E1 13320.648,E2 13320.648} C_VEL
LIN {X 0,Y 442.431,Z 470.407,A -85,B 0,C 180,E1 13315.983,E2 13315.983} C_VEL
LIN {X 0,Y 444.381,Z 474.753,A -85,B 0,C 180,E1 13311.981,E2 13311.981} C_VEL
LIN {X 0,Y 445.232,Z 475.892,A -85,B 0,C 180,E1 13310.955,E2 13310.955} C_VEL
LIN {X 0,Y 448.022,Z 480.655,A -85,B 0,C 180,E1 13308.217,E2 13308.217} C_VEL
LIN {X 0,Y 451.114,Z 485.783,A -85,B 0,C 180,E1 13305.888,E2 13305.888} C_VEL
LIN {X 0,Y 455.076,Z 492.534,A -85,B 0,C 180,E1 13303.436,E2 13303.436} C_VEL
LIN {X 0,Y 458.741,Z 499.273,A -85,B 0,C 180,E1 13301.477,E2 13301.477} C_VEL
LIN {X 0,Y 439.184,Z 716.37,A -85,B 0,C 180,E1 13298.152,E2 13298.152} C_VEL
LIN {X 0,Y 435.488,Z 742.663,A -85,B 0,C 180,E1 13297.669,E2 13297.669} C_VEL
LIN {X 0,Y 430.416,Z 767.563,A -85,B 0,C 180,E1 13297.077,E2 13297.077} C_VEL
LIN {X 0,Y 425.651,Z 786.854,A -85,B 0,C 180,E1 13296.499,E2 13296.499} C_VEL
LIN {X 0,Y 418.897,Z 810.119,A -85,B 0,C 180,E1 13295.648,E2 13295.648} C_VEL
LIN {X 0,Y 410.495,Z 834.375,A -85,B 0,C 180,E1 13294.531,E2 13294.531} C_VEL
LIN {X 0,Y 402.565,Z 854.538,A -85,B 0,C 180,E1 13293.401,E2 13293.401} C_VEL
LIN {X 0,Y 393.119,Z 876.164,A -85,B 0,C 180,E1 13291.956,E2 13291.956} C_VEL
LIN {X 0,Y 382.524,Z 897.606,A -85,B 0,C 180,E1 13290.206,E2 13290.206} C_VEL
LIN {X 0,Y 373.322,Z 914.765,A -85,B 0,C 180,E1 13288.545,E2 13288.545} C_VEL
LIN {X 0,Y 362.847,Z 932.989,A -85,B 0,C 180,E1 13286.469,E2 13286.469} C_VEL
LIN {X 0,Y 351.237,Z 951.663,A -85,B 0,C 180,E1 13283.894,E2 13283.894} C_VEL
LIN {X 0,Y 341.423,Z 966.58,A -85,B 0,C 180,E1 13281.438,E2 13281.438} C_VEL
LIN {X 0,Y 331.632,Z 980.915,A -85,B 0,C 180,E1 13278.655,E2 13278.655} C_VEL
LIN {X 0,Y 320.193,Z 997.043,A -85,B 0,C 180,E1 13274.857,E2 13274.857} C_VEL
LIN {X 0,Y 311.469,Z 1009.107,A -85,B 0,C 180,E1 13271.399,E2 13271.399} C_VEL
LIN {X 0,Y 302.946,Z 1021.053,A -85,B 0,C 180,E1 13267.303,E2 13267.303} C_VEL
LIN {X 0,Y 295.176,Z 1032.112,A -85,B 0,C 180,E1 13262.588,E2 13262.588} C_VEL
LIN {X 0,Y 289.946,Z 1040.111,A -85,B 0,C 180,E1 13258.418,E2 13258.418} C_VEL
LIN {X 0,Y 285.302,Z 1048.081,A -85,B 0,C 180,E1 13253.33,E2 13253.33} C_VEL
LIN {X 0,Y 282.275,Z 1054.153,A -85,B 0,C 180,E1 13248.163,E2 13248.163} C_VEL
LIN {X 0,Y 280.864,Z 1057.901,A -85,B 0,C 180,E1 13244.01,E2 13244.01} C_VEL
LIN {X 0,Y 280.159,Z 1060.636,A -85,B 0,C 180,E1 13239.864,E2 13239.864} C_VEL
LIN {X 0,Y 279.932,Z 1062.306,A -85,B 0,C 180,E1 13235.946,E2 13235.946} C_VEL
LIN {X 0,Y 279.907,Z 1063.078,A -85,B 0,C 180,E1 13232.047,E2 13232.047} C_VEL
LIN {X 0,Y 279.907,Z 1062.948,A -85,B 0,C 180,E1 13228.158,E2 13228.158} C_VEL
LIN {X 0,Y 279.94,Z 1061.776,A -85,B 0,C 180,E1 13223.849,E2 13223.849} C_VEL
LIN {X 0,Y 280.288,Z 1059.043,A -85,B 0,C 180,E1 13218.893,E2 13218.893} C_VEL
LIN {X 0,Y 281.286,Z 1055.173,A -85,B 0,C 180,E1 13214.327,E2 13214.327} C_VEL
LIN {X 0,Y 283.084,Z 1050.31,A -85,B 0,C 180,E1 13209.964,E2 13209.964} C_VEL
LIN {X 0,Y 286.243,Z 1043.641,A -85,B 0,C 180,E1 13205.218,E2 13205.218} C_VEL
LIN {X 0,Y 291.253,Z 1034.55,A -85,B 0,C 180,E1 13200.146,E2 13200.146} C_VEL
LIN {X 0,Y 296.529,Z 1025.892,A -85,B 0,C 180,E1 13196.195,E2 13196.195} C_VEL
LIN {X 0,Y 303.263,Z 1015.409,A -85,B 0,C 180,E1 13192.175,E2 13192.175} C_VEL
LIN {X 0,Y 312.493,Z 1001.388,A -85,B 0,C 180,E1 13187.783,E2 13187.783} C_VEL
LIN {X 0,Y 320.887,Z 988.618,A -85,B 0,C 180,E1 13184.474,E2 13184.474} C_VEL
LIN {X 0,Y 330.729,Z 973.487,A -85,B 0,C 180,E1 13181.167,E2 13181.167} C_VEL
LIN {X 0,Y 341.528,Z 956.055,A -85,B 0,C 180,E1 13178.043,E2 13178.043} C_VEL
LIN {X 0,Y 350.823,Z 940.389,A -85,B 0,C 180,E1 13175.681,E2 13175.681} C_VEL
LIN {X 0,Y 361.63,Z 921.228,A -85,B 0,C 180,E1 13173.239,E2 13173.239} C_VEL
LIN {X 0,Y 372.012,Z 900.996,A -85,B 0,C 180,E1 13171.124,E2 13171.124} C_VEL
LIN {X 0,Y 380.655,Z 882.858,A -85,B 0,C 180,E1 13169.517,E2 13169.517} C_VEL
LIN {X 0,Y 390.61,Z 860.004,A -85,B 0,C 180,E1 13167.821,E2 13167.821} C_VEL
LIN {X 0,Y 398.99,Z 838.078,A -85,B 0,C 180,E1 13166.492,E2 13166.492} C_VEL
LIN {X 0,Y 405.738,Z 818.313,A -85,B 0,C 180,E1 13165.489,E2 13165.489} C_VEL
LIN {X 0,Y 413.15,Z 793.372,A -85,B 0,C 180,E1 13164.447,E2 13164.447} C_VEL
LIN {X 0,Y 418.877,Z 769.715,A -85,B 0,C 180,E1 13163.668,E2 13163.668} C_VEL
LIN {X 0,Y 423.304,Z 747.615,A -85,B 0,C 180,E1 13163.099,E2 13163.099} C_VEL
LIN {X 0,Y 427.418,Z 719.607,A -85,B 0,C 180,E1 13162.539,E2 13162.539} C_VEL
LIN {X 0,Y 433.358,Z 651.148,A -85,B 0,C 180,E1 13161.444,E2 13161.444} C_VEL
LIN {X 0,Y 446.854,Z 491.031,A -85,B 0,C 180,E1 13158.933,E2 13158.933} C_VEL
LIN {X 0,Y 443.397,Z 484.6,A -85,B 0,C 180,E1 13157.385,E2 13157.385} C_VEL
LIN {X 0,Y 437.99,Z 475.483,A -85,B 0,C 180,E1 13154.679,E2 13154.679} C_VEL
LIN {X 0,Y 433.686,Z 468.389,A -85,B 0,C 180,E1 13152.111,E2 13152.111} C_VEL
LIN {X 0,Y 430.838,Z 463.862,A -85,B 0,C 180,E1 13150.092,E2 13150.092} C_VEL
LIN {X 0,Y 428.311,Z 459.778,A -85,B 0,C 180,E1 13147.917,E2 13147.917} C_VEL
LIN {X 0,Y 425.579,Z 455.219,A -85,B 0,C 180,E1 13144.717,E2 13144.717} C_VEL
LIN {X 0,Y 423.42,Z 451.94,A -85,B 0,C 180,E1 13138.647,E2 13138.647} C_VEL
LIN {X 0,Y 423.688,Z 452.913,A -85,B 0,C 180,E1 13135.94,E2 13135.94} C_VEL
LIN {X 0,Y 425.862,Z 455.701,A -85,B 0,C 180,E1 13131.698,E2 13131.698} C_VEL
LIN {X 0,Y 429.033,Z 460.938,A -85,B 0,C 180,E1 13128.233,E2 13128.233} C_VEL
LIN {X 0,Y 432.087,Z 465.839,A -85,B 0,C 180,E1 13125.801,E2 13125.801} C_VEL
LIN {X 0,Y 435.451,Z 471.336,A -85,B 0,C 180,E1 13123.594,E2 13123.594} C_VEL
LIN {X 0,Y 439.659,Z 478.155,A -85,B 0,C 180,E1 13121.262,E2 13121.262} C_VEL
LIN {X 0,Y 446.326,Z 489.654,A -85,B 0,C 180,E1 13118.133,E2 13118.133} C_VEL
LIN {X 0,Y 446.871,Z 490.993,A -85,B 0,C 180,E1 13117.883,E2 13117.883} C_VEL
LIN {X 0,Y 428.001,Z 712.557,A -85,B 0,C 180,E1 13114.419,E2 13114.419} C_VEL
LIN {X 0,Y 424.574,Z 738.505,A -85,B 0,C 180,E1 13113.925,E2 13113.925} C_VEL
LIN {X 0,Y 419.647,Z 763.962,A -85,B 0,C 180,E1 13113.279,E2 13113.279} C_VEL
LIN {X 0,Y 414.556,Z 785.566,A -85,B 0,C 180,E1 13112.572,E2 13112.572} C_VEL
LIN {X 0,Y 407.488,Z 810.593,A -85,B 0,C 180,E1 13111.557,E2 13111.557} C_VEL
LIN {X 0,Y 400.394,Z 831.79,A -85,B 0,C 180,E1 13110.492,E2 13110.492} C_VEL
LIN {X 0,Y 393.318,Z 850.627,A -85,B 0,C 180,E1 13109.376,E2 13109.376} C_VEL
LIN {X 0,Y 384.029,Z 872.982,A -85,B 0,C 180,E1 13107.8,E2 13107.8} C_VEL
LIN {X 0,Y 374.031,Z 894.232,A -85,B 0,C 180,E1 13105.966,E2 13105.966} C_VEL
LIN {X 0,Y 365.053,Z 911.863,A -85,B 0,C 180,E1 13104.169,E2 13104.169} C_VEL
LIN {X 0,Y 354.345,Z 931.488,A -85,B 0,C 180,E1 13101.801,E2 13101.801} C_VEL
LIN {X 0,Y 343.655,Z 949.488,A -85,B 0,C 180,E1 13099.155,E2 13099.155} C_VEL
LIN {X 0,Y 334.302,Z 964.565,A -85,B 0,C 180,E1 13096.534,E2 13096.534} C_VEL
LIN {X 0,Y 323.118,Z 981.88,A -85,B 0,C 180,E1 13092.905,E2 13092.905} C_VEL
LIN {X 0,Y 314.676,Z 994.54,A -85,B 0,C 180,E1 13089.693,E2 13089.693} C_VEL
LIN {X 0,Y 306.782,Z 1006.359,A -85,B 0,C 180,E1 13086.152,E2 13086.152} C_VEL
LIN {X 0,Y 298.094,Z 1019.526,A -85,B 0,C 180,E1 13081.326,E2 13081.326} C_VEL
LIN {X 0,Y 292.323,Z 1028.655,A -85,B 0,C 180,E1 13077.21,E2 13077.21} C_VEL
LIN {X 0,Y 287.358,Z 1037.285,A -85,B 0,C 180,E1 13072.504,E2 13072.504} C_VEL
LIN {X 0,Y 283.661,Z 1044.532,A -85,B 0,C 180,E1 13067.435,E2 13067.435} C_VEL
LIN {X 0,Y 281.687,Z 1049.369,A -85,B 0,C 180,E1 13063.131,E2 13063.131} C_VEL
LIN {X 0,Y 280.55,Z 1053.092,A -85,B 0,C 180,E1 13058.815,E2 13058.815} C_VEL
LIN {X 0,Y 280.021,Z 1056.069,A -85,B 0,C 180,E1 13053.89,E2 13053.89} C_VEL
LIN {X 0,Y 279.918,Z 1057.461,A -85,B 0,C 180,E1 13049.181,E2 13049.181} C_VEL
LIN {X 0,Y 279.913,Z 1057.658,A -85,B 0,C 180,E1 13045.082,E2 13045.082} C_VEL
LIN {X 0,Y 279.976,Z 1056.95,A -85,B 0,C 180,E1 13041.166,E2 13041.166} C_VEL
LIN {X 0,Y 280.259,Z 1055.349,A -85,B 0,C 180,E1 13037.221,E2 13037.221} C_VEL
LIN {X 0,Y 281.054,Z 1052.681,A -85,B 0,C 180,E1 13033.039,E2 13033.039} C_VEL
LIN {X 0,Y 282.671,Z 1048.783,A -85,B 0,C 180,E1 13028.633,E2 13028.633} C_VEL
LIN {X 0,Y 286.082,Z 1042.344,A -85,B 0,C 180,E1 13023.201,E2 13023.201} C_VEL
LIN {X 0,Y 290.616,Z 1034.968,A -85,B 0,C 180,E1 13018.468,E2 13018.468} C_VEL
LIN {X 0,Y 296.074,Z 1026.918,A -85,B 0,C 180,E1 13014.25,E2 13014.25} C_VEL
LIN {X 0,Y 304.636,Z 1014.964,A -85,B 0,C 180,E1 13009.219,E2 13009.219} C_VEL
LIN {X 0,Y 312.578,Z 1004.085,A -85,B 0,C 180,E1 13005.508,E2 13005.508} C_VEL
LIN {X 0,Y 322.058,Z 991.189,A -85,B 0,C 180,E1 13001.83,E2 13001.83} C_VEL
LIN {X 0,Y 332.734,Z 976.202,A -85,B 0,C 180,E1 12998.342,E2 12998.342} C_VEL
LIN {X 0,Y 342.174,Z 962.493,A -85,B 0,C 180,E1 12995.673,E2 12995.673} C_VEL
LIN {X 0,Y 352.285,Z 947.201,A -85,B 0,C 180,E1 12993.145,E2 12993.145} C_VEL
LIN {X 0,Y 364.687,Z 927.17,A -85,B 0,C 180,E1 12990.407,E2 12990.407} C_VEL
LIN {X 0,Y 374.328,Z 910.387,A -85,B 0,C 180,E1 12988.501,E2 12988.501} C_VEL
LIN {X 0,Y 384.044,Z 892.219,A -85,B 0,C 180,E1 12986.744,E2 12986.744} C_VEL
LIN {X 0,Y 395.19,Z 869.184,A -85,B 0,C 180,E1 12984.899,E2 12984.899} C_VEL
LIN {X 0,Y 403.703,Z 849.518,A -85,B 0,C 180,E1 12983.593,E2 12983.593} C_VEL
LIN {X 0,Y 412.425,Z 827.074,A -85,B 0,C 180,E1 12982.345,E2 12982.345} C_VEL
LIN {X 0,Y 417.285,Z 812.909,A -85,B 0,C 180,E1 12981.686,E2 12981.686} C_VEL
LIN {X 0,Y 418.977,Z 806.998,A -85,B 0,C 180,E1 12981.336,E2 12981.336} C_VEL
LIN {X 0,Y 422.142,Z 788.038,A -85,B 0,C 180,E1 12979.789,E2 12979.789} C_VEL
LIN {X 0,Y 423.472,Z 781.934,A -85,B 0,C 180,E1 12979.485,E2 12979.485} C_VEL
LIN {X 0,Y 429.009,Z 759.211,A -85,B 0,C 180,E1 12978.818,E2 12978.818} C_VEL
LIN {X 0,Y 433.981,Z 732.733,A -85,B 0,C 180,E1 12978.228,E2 12978.228} C_VEL
LIN {X 0,Y 436.978,Z 710.315,A -85,B 0,C 180,E1 12977.833,E2 12977.833} C_VEL
LIN {X 0,Y 455.904,Z 504.336,A -85,B 0,C 180,E1 12974.702,E2 12974.702} C_VEL
LIN {X 0,Y 451.022,Z 495.567,A -85,B 0,C 180,E1 12971.834,E2 12971.834} C_VEL
LIN {X 0,Y 447.847,Z 490.33,A -85,B 0,C 180,E1 12969.575,E2 12969.575} C_VEL
LIN {X 0,Y 445.873,Z 486.864,A -85,B 0,C 180,E1 12967.862,E2 12967.862} C_VEL
LIN {X 0,Y 443.556,Z 482.819,A -85,B 0,C 180,E1 12965.303,E2 12965.303} C_VEL
LIN {X 0,Y 441.451,Z 478.55,A -85,B 0,C 180,E1 12961.168,E2 12961.168} C_VEL
LIN {X 0,Y 441.047,Z 478.065,A -85,B 0,C 180,E1 12958.441,E2 12958.441} C_VEL
LIN {X 0,Y 441.444,Z 478.461,A -85,B 0,C 180,E1 12955.974,E2 12955.974} C_VEL
LIN {X 0,Y 443.409,Z 482.74,A -85,B 0,C 180,E1 12951.963,E2 12951.963} C_VEL
LIN {X 0,Y 444.189,Z 483.942,A -85,B 0,C 180,E1 12950.999,E2 12950.999} C_VEL
LIN {X 0,Y 446.74,Z 488.353,A -85,B 0,C 180,E1 12948.444,E2 12948.444} C_VEL
LIN {X 0,Y 449.758,Z 493.492,A -85,B 0,C 180,E1 12946.107,E2 12946.107} C_VEL
LIN {X 0,Y 453.639,Z 500.315,A -85,B 0,C 180,E1 12943.645,E2 12943.645} C_VEL
LIN {X 0,Y 455.938,Z 504.682,A -85,B 0,C 180,E1 12942.358,E2 12942.358} C_VEL
LIN {X 0,Y 436.367,Z 717.017,A -85,B 0,C 180,E1 12939.129,E2 12939.129} C_VEL
LIN {X 0,Y 432.422,Z 743.931,A -85,B 0,C 180,E1 12938.634,E2 12938.634} C_VEL
LIN {X 0,Y 427.459,Z 767.8,A -85,B 0,C 180,E1 12938.071,E2 12938.071} C_VEL
LIN {X 0,Y 422.542,Z 787.299,A -85,B 0,C 180,E1 12937.496,E2 12937.496} C_VEL
LIN {X 0,Y 415.135,Z 812.211,A -85,B 0,C 180,E1 12936.587,E2 12936.587} C_VEL
LIN {X 0,Y 406.603,Z 835.986,A -85,B 0,C 180,E1 12935.488,E2 12935.488} C_VEL
LIN {X 0,Y 398.64,Z 855.714,A -85,B 0,C 180,E1 12934.384,E2 12934.384} C_VEL
LIN {X 0,Y 388.27,Z 878.648,A -85,B 0,C 180,E1 12932.841,E2 12932.841} C_VEL
LIN {X 0,Y 378.19,Z 898.456,A -85,B 0,C 180,E1 12931.216,E2 12931.216} C_VEL
LIN {X 0,Y 368.782,Z 915.532,A -85,B 0,C 180,E1 12929.564,E2 12929.564} C_VEL
LIN {X 0,Y 357.008,Z 935.406,A -85,B 0,C 180,E1 12927.279,E2 12927.279} C_VEL
LIN {X 0,Y 345.947,Z 952.512,A -85,B 0,C 180,E1 12924.88,E2 12924.88} C_VEL
LIN {X 0,Y 336.331,Z 966.668,A -85,B 0,C 180,E1 12922.539,E2 12922.539} C_VEL
LIN {X 0,Y 325.679,Z 981.755,A -85,B 0,C 180,E1 12919.588,E2 12919.588} C_VEL
LIN {X 0,Y 313.938,Z 997.64,A -85,B 0,C 180,E1 12915.776,E2 12915.776} C_VEL
LIN {X 0,Y 305.28,Z 1009.139,A -85,B 0,C 180,E1 12912.432,E2 12912.432} C_VEL
LIN {X 0,Y 295.995,Z 1021.596,A -85,B 0,C 180,E1 12908.085,E2 12908.085} C_VEL
LIN {X 0,Y 287.91,Z 1032.516,A -85,B 0,C 180,E1 12903.279,E2 12903.279} C_VEL
LIN {X 0,Y 282.447,Z 1040.453,A -85,B 0,C 180,E1 12899.012,E2 12899.012} C_VEL
LIN {X 0,Y 277.414,Z 1048.574,A -85,B 0,C 180,E1 12893.583,E2 12893.583} C_VEL
LIN {X 0,Y 274.484,Z 1054.113,A -85,B 0,C 180,E1 12888.697,E2 12888.697} C_VEL
LIN {X 0,Y 272.96,Z 1057.852,A -85,B 0,C 180,E1 12884.424,E2 12884.424} C_VEL
LIN {X 0,Y 272.182,Z 1060.614,A -85,B 0,C 180,E1 12880.091,E2 12880.091} C_VEL
LIN {X 0,Y 271.931,Z 1062.31,A -85,B 0,C 180,E1 12875.909,E2 12875.909} C_VEL
LIN {X 0,Y 271.908,Z 1063.073,A -85,B 0,C 180,E1 12871.475,E2 12871.475} C_VEL
LIN {X 0,Y 271.912,Z 1062.716,A -85,B 0,C 180,E1 12866.838,E2 12866.838} C_VEL
LIN {X 0,Y 272.028,Z 1060.906,A -85,B 0,C 180,E1 12861.971,E2 12861.971} C_VEL
LIN {X 0,Y 272.505,Z 1058.125,A -85,B 0,C 180,E1 12857.497,E2 12857.497} C_VEL
LIN {X 0,Y 273.637,Z 1054.415,A -85,B 0,C 180,E1 12853.211,E2 12853.211} C_VEL
LIN {X 0,Y 275.848,Z 1049.148,A -85,B 0,C 180,E1 12848.525,E2 12848.525} C_VEL
LIN {X 0,Y 280.056,Z 1041.118,A -85,B 0,C 180,E1 12843.036,E2 12843.036} C_VEL
LIN {X 0,Y 284.831,Z 1033.158,A -85,B 0,C 180,E1 12838.698,E2 12838.698} C_VEL
LIN {X 0,Y 290.87,Z 1023.86,A -85,B 0,C 180,E1 12834.483,E2 12834.483} C_VEL
LIN {X 0,Y 299.753,Z 1010.778,A -85,B 0,C 180,E1 12829.675,E2 12829.675} C_VEL
LIN {X 0,Y 307.72,Z 999.16,A -85,B 0,C 180,E1 12826.167,E2 12826.167} C_VEL
LIN {X 0,Y 317.127,Z 985.439,A -85,B 0,C 180,E1 12822.679,E2 12822.679} C_VEL
LIN {X 0,Y 328.003,Z 969.043,A -85,B 0,C 180,E1 12819.259,E2 12819.259} C_VEL
LIN {X 0,Y 337.638,Z 953.915,A -85,B 0,C 180,E1 12816.627,E2 12816.627} C_VEL
LIN {X 0,Y 348.55,Z 936.004,A -85,B 0,C 180,E1 12813.999,E2 12813.999} C_VEL
LIN {X 0,Y 359.737,Z 916.067,A -85,B 0,C 180,E1 12811.601,E2 12811.601} C_VEL
LIN {X 0,Y 368.844,Z 898.62,A -85,B 0,C 180,E1 12809.834,E2 12809.834} C_VEL
LIN {X 0,Y 379.314,Z 876.946,A -85,B 0,C 180,E1 12807.984,E2 12807.984} C_VEL
LIN {X 0,Y 388.664,Z 855.014,A -85,B 0,C 180,E1 12806.457,E2 12806.457} C_VEL
LIN {X 0,Y 396.048,Z 835.838,A -85,B 0,C 180,E1 12805.335,E2 12805.335} C_VEL
LIN {X 0,Y 403.928,Z 812.899,A -85,B 0,C 180,E1 12804.216,E2 12804.216} C_VEL
LIN {X 0,Y 410.89,Z 788.674,A -85,B 0,C 180,E1 12803.274,E2 12803.274} C_VEL
LIN {X 0,Y 415.891,Z 768.048,A -85,B 0,C 180,E1 12802.621,E2 12802.621} C_VEL
LIN {X 0,Y 420.685,Z 744.096,A -85,B 0,C 180,E1 12802.024,E2 12802.024} C_VEL
LIN {X 0,Y 424.464,Z 717.215,A -85,B 0,C 180,E1 12801.508,E2 12801.508} C_VEL
LIN {X 0,Y 442.908,Z 505.535,A -85,B 0,C 180,E1 12798.21,E2 12798.21} C_VEL
LIN {X 0,Y 443.72,Z 495.913,A -85,B 0,C 180,E1 12798.05,E2 12798.05} C_VEL
LIN {X 0,Y 438.832,Z 487.178,A -85,B 0,C 180,E1 12795.699,E2 12795.699} C_VEL
LIN {X 0,Y 433.997,Z 478.977,A -85,B 0,C 180,E1 12792.981,E2 12792.981} C_VEL
LIN {X 0,Y 430.03,Z 472.218,A -85,B 0,C 180,E1 12790.246,E2 12790.246} C_VEL
LIN {X 0,Y 427.047,Z 467.495,A -85,B 0,C 180,E1 12787.67,E2 12787.67} C_VEL
LIN {X 0,Y 424.407,Z 463.037,A -85,B 0,C 180,E1 12784.459,E2 12784.459} C_VEL
LIN {X 0,Y 422.445,Z 459.855,A -85,B 0,C 180,E1 12778.508,E2 12778.508} C_VEL
LIN {X 0,Y 422.817,Z 461.159,A -85,B 0,C 180,E1 12775.524,E2 12775.524} C_VEL
LIN {X 0,Y 424.74,Z 463.515,A -85,B 0,C 180,E1 12771.88,E2 12771.88} C_VEL
LIN {X 0,Y 427.758,Z 468.636,A -85,B 0,C 180,E1 12768.471,E2 12768.471} C_VEL
LIN {X 0,Y 430.737,Z 473.552,A -85,B 0,C 180,E1 12766.03,E2 12766.03} C_VEL
LIN {X 0,Y 434.14,Z 479.232,A -85,B 0,C 180,E1 12763.75,E2 12763.75} C_VEL
LIN {X 0,Y 438.408,Z 486.389,A -85,B 0,C 180,E1 12761.345,E2 12761.345} C_VEL
LIN {X 0,Y 443.702,Z 495.879,A -85,B 0,C 180,E1 12758.779,E2 12758.779} C_VEL
LIN {X 0,Y 424.715,Z 713.534,A -85,B 0,C 180,E1 12755.392,E2 12755.392} C_VEL
LIN {X 0,Y 421.071,Z 739.935,A -85,B 0,C 180,E1 12754.887,E2 12754.887} C_VEL
LIN {X 0,Y 416.202,Z 764.498,A -85,B 0,C 180,E1 12754.266,E2 12754.266} C_VEL
LIN {X 0,Y 410.947,Z 786.309,A -85,B 0,C 180,E1 12753.558,E2 12753.558} C_VEL
LIN {X 0,Y 403.487,Z 811.95,A -85,B 0,C 180,E1 12752.519,E2 12752.519} C_VEL
LIN {X 0,Y 396.51,Z 832.327,A -85,B 0,C 180,E1 12751.5,E2 12751.5} C_VEL
LIN {X 0,Y 388.935,Z 852.007,A -85,B 0,C 180,E1 12750.335,E2 12750.335} C_VEL
LIN {X 0,Y 379.104,Z 874.888,A -85,B 0,C 180,E1 12748.71,E2 12748.71} C_VEL
LIN {X 0,Y 369.236,Z 895.279,A -85,B 0,C 180,E1 12746.942,E2 12746.942} C_VEL
LIN {X 0,Y 360.051,Z 912.825,A -85,B 0,C 180,E1 12745.147,E2 12745.147} C_VEL
LIN {X 0,Y 348.455,Z 933.306,A -85,B 0,C 180,E1 12742.641,E2 12742.641} C_VEL
LIN {X 0,Y 338.382,Z 949.784,A -85,B 0,C 180,E1 12740.199,E2 12740.199} C_VEL
LIN {X 0,Y 328.923,Z 964.559,A -85,B 0,C 180,E1 12737.62,E2 12737.62} C_VEL
LIN {X 0,Y 317.652,Z 981.435,A -85,B 0,C 180,E1 12734.079,E2 12734.079} C_VEL
LIN {X 0,Y 308.361,Z 994.849,A -85,B 0,C 180,E1 12730.644,E2 12730.644} C_VEL
LIN {X 0,Y 300.206,Z 1006.575,A -85,B 0,C 180,E1 12727.074,E2 12727.074} C_VEL
LIN {X 0,Y 291.434,Z 1019.264,A -85,B 0,C 180,E1 12722.359,E2 12722.359} C_VEL
LIN {X 0,Y 285.408,Z 1028.307,A -85,B 0,C 180,E1 12718.226,E2 12718.226} C_VEL
LIN {X 0,Y 280.413,Z 1036.405,A -85,B 0,C 180,E1 12713.761,E2 12713.761} C_VEL
LIN {X 0,Y 276.039,Z 1044.421,A -85,B 0,C 180,E1 12708.15,E2 12708.15} C_VEL
LIN {X 0,Y 273.886,Z 1049.293,A -85,B 0,C 180,E1 12703.727,E2 12703.727} C_VEL
LIN {X 0,Y 272.661,Z 1052.94,A -85,B 0,C 180,E1 12699.436,E2 12699.436} C_VEL
LIN {X 0,Y 272.078,Z 1055.725,A -85,B 0,C 180,E1 12694.849,E2 12694.849} C_VEL
LIN {X 0,Y 271.939,Z 1057.477,A -85,B 0,C 180,E1 12689.789,E2 12689.789} C_VEL
LIN {X 0,Y 271.913,Z 1057.753,A -85,B 0,C 180,E1 12685.148,E2 12685.148} C_VEL
LIN {X 0,Y 271.987,Z 1057.012,A -85,B 0,C 180,E1 12680.905,E2 12680.905} C_VEL
LIN {X 0,Y 272.309,Z 1055.401,A -85,B 0,C 180,E1 12676.841,E2 12676.841} C_VEL
LIN {X 0,Y 273.186,Z 1052.722,A -85,B 0,C 180,E1 12672.535,E2 12672.535} C_VEL
LIN {X 0,Y 274.927,Z 1048.846,A -85,B 0,C 180,E1 12668.036,E2 12668.036} C_VEL
LIN {X 0,Y 278.644,Z 1042.341,A -85,B 0,C 180,E1 12662.418,E2 12662.418} C_VEL
LIN {X 0,Y 283.483,Z 1034.962,A -85,B 0,C 180,E1 12657.58,E2 12657.58} C_VEL
LIN {X 0,Y 289.266,Z 1026.9,A -85,B 0,C 180,E1 12653.273,E2 12653.273} C_VEL
LIN {X 0,Y 298.281,Z 1014.919,A -85,B 0,C 180,E1 12648.158,E2 12648.158} C_VEL
LIN {X 0,Y 306.571,Z 1004.074,A -85,B 0,C 180,E1 12644.417,E2 12644.417} C_VEL
LIN {X 0,Y 317.006,Z 990.478,A -85,B 0,C 180,E1 12640.523,E2 12640.523} C_VEL
LIN {X 0,Y 328.132,Z 975.321,A -85,B 0,C 180,E1 12637.026,E2 12637.026} C_VEL
LIN {X 0,Y 337.94,Z 961.519,A -85,B 0,C 180,E1 12634.361,E2 12634.361} C_VEL
LIN {X 0,Y 349.773,Z 944.133,A -85,B 0,C 180,E1 12631.543,E2 12631.543} C_VEL
LIN {X 0,Y 361.499,Z 925.375,A -85,B 0,C 180,E1 12629.069,E2 12629.069} C_VEL
LIN {X 0,Y 371.137,Z 908.952,A -85,B 0,C 180,E1 12627.245,E2 12627.245} C_VEL
LIN {X 0,Y 382.219,Z 888.6,A -85,B 0,C 180,E1 12625.334,E2 12625.334} C_VEL
LIN {X 0,Y 392.17,Z 868.067,A -85,B 0,C 180,E1 12623.75,E2 12623.75} C_VEL
LIN {X 0,Y 400.488,Z 849.18,A -85,B 0,C 180,E1 12622.517,E2 12622.517} C_VEL
LIN {X 0,Y 409.383,Z 826.688,A -85,B 0,C 180,E1 12621.286,E2 12621.286} C_VEL
LIN {X 0,Y 417.653,Z 802.064,A -85,B 0,C 180,E1 12620.204,E2 12620.204} C_VEL
LIN {X 0,Y 423.472,Z 781.934,A -85,B 0,C 180,E1 12619.485,E2 12619.485} C_VEL
LIN {X 0,Y 425.074,Z 774.78,A -85,B 0,C 180,E1 12619.135,E2 12619.135} C_VEL
LIN {X 0,Y 427.134,Z 757.077,A -85,B 0,C 180,E1 12617.878,E2 12617.878} C_VEL
LIN {X 0,Y 428.247,Z 749.751,A -85,B 0,C 180,E1 12617.582,E2 12617.582} C_VEL
LIN {X 0,Y 432.023,Z 728.347,A -85,B 0,C 180,E1 12617.144,E2 12617.144} C_VEL
LIN {X 0,Y 435.31,Z 701.932,A -85,B 0,C 180,E1 12616.699,E2 12616.699} C_VEL
LIN {X 0,Y 453.194,Z 509.868,A -85,B 0,C 180,E1 12613.808,E2 12613.808} C_VEL
LIN {X 0,Y 449.166,Z 502.522,A -85,B 0,C 180,E1 12611.297,E2 12611.297} C_VEL
LIN {X 0,Y 446.536,Z 498.012,A -85,B 0,C 180,E1 12609.343,E2 12609.343} C_VEL
LIN {X 0,Y 444.614,Z 494.565,A -85,B 0,C 180,E1 12607.625,E2 12607.625} C_VEL
LIN {X 0,Y 442.474,Z 490.697,A -85,B 0,C 180,E1 12605.186,E2 12605.186} C_VEL
LIN {X 0,Y 440.438,Z 486.43,A -85,B 0,C 180,E1 12601.041,E2 12601.041} C_VEL
LIN {X 0,Y 440.108,Z 486.016,A -85,B 0,C 180,E1 12597.787,E2 12597.787} C_VEL
LIN {X 0,Y 440.458,Z 486.513,A -85,B 0,C 180,E1 12595.965,E2 12595.965} C_VEL
LIN {X 0,Y 442.438,Z 490.726,A -85,B 0,C 180,E1 12591.945,E2 12591.945} C_VEL
LIN {X 0,Y 443.306,Z 492.323,A -85,B 0,C 180,E1 12590.85,E2 12590.85} C_VEL
LIN {X 0,Y 445.464,Z 496.051,A -85,B 0,C 180,E1 12588.673,E2 12588.673} C_VEL
LIN {X 0,Y 448.409,Z 501.2,A -85,B 0,C 180,E1 12586.328,E2 12586.328} C_VEL
LIN {X 0,Y 452.312,Z 508.293,A -85,B 0,C 180,E1 12583.794,E2 12583.794} C_VEL
LIN {X 0,Y 453.241,Z 510.094,A -85,B 0,C 180,E1 12583.251,E2 12583.251} C_VEL
LIN {X 0,Y 433.762,Z 716.927,A -85,B 0,C 180,E1 12580.13,E2 12580.13} C_VEL
LIN {X 0,Y 429.765,Z 743.78,A -85,B 0,C 180,E1 12579.643,E2 12579.643} C_VEL
LIN {X 0,Y 424.722,Z 767.671,A -85,B 0,C 180,E1 12579.089,E2 12579.089} C_VEL
LIN {X 0,Y 419.792,Z 786.917,A -85,B 0,C 180,E1 12578.533,E2 12578.533} C_VEL
LIN {X 0,Y 412.498,Z 811.138,A -85,B 0,C 180,E1 12577.672,E2 12577.672} C_VEL
LIN {X 0,Y 403.721,Z 835.31,A -85,B 0,C 180,E1 12576.579,E2 12576.579} C_VEL
LIN {X 0,Y 395.604,Z 855.1,A -85,B 0,C 180,E1 12575.491,E2 12575.491} C_VEL
LIN {X 0,Y 385.393,Z 877.403,A -85,B 0,C 180,E1 12574.024,E2 12574.024} C_VEL
LIN {X 0,Y 374.702,Z 897.982,A -85,B 0,C 180,E1 12572.367,E2 12572.367} C_VEL
LIN {X 0,Y 364.71,Z 915.697,A -85,B 0,C 180,E1 12570.671,E2 12570.671} C_VEL
LIN {X 0,Y 352.375,Z 935.922,A -85,B 0,C 180,E1 12568.35,E2 12568.35} C_VEL
LIN {X 0,Y 340.908,Z 953.148,A -85,B 0,C 180,E1 12565.93,E2 12565.93} C_VEL
LIN {X 0,Y 330.176,Z 968.441,A -85,B 0,C 180,E1 12563.37,E2 12563.37} C_VEL
LIN {X 0,Y 317.615,Z 985.479,A -85,B 0,C 180,E1 12559.906,E2 12559.906} C_VEL
LIN {X 0,Y 307.206,Z 998.952,A -85,B 0,C 180,E1 12556.537,E2 12556.537} C_VEL
LIN {X 0,Y 297.861,Z 1010.889,A -85,B 0,C 180,E1 12552.957,E2 12552.957} C_VEL
LIN {X 0,Y 287.768,Z 1023.743,A -85,B 0,C 180,E1 12548.206,E2 12548.206} C_VEL
LIN {X 0,Y 280.688,Z 1032.92,A -85,B 0,C 180,E1 12544.006,E2 12544.006} C_VEL
LIN {X 0,Y 274.738,Z 1041.149,A -85,B 0,C 180,E1 12539.428,E2 12539.428} C_VEL
LIN {X 0,Y 269.369,Z 1049.309,A -85,B 0,C 180,E1 12533.634,E2 12533.634} C_VEL
LIN {X 0,Y 266.612,Z 1054.28,A -85,B 0,C 180,E1 12529.043,E2 12529.043} C_VEL
LIN {X 0,Y 265.007,Z 1057.964,A -85,B 0,C 180,E1 12524.643,E2 12524.643} C_VEL
LIN {X 0,Y 264.174,Z 1060.751,A -85,B 0,C 180,E1 12520.027,E2 12520.027} C_VEL
LIN {X 0,Y 263.916,Z 1062.52,A -85,B 0,C 180,E1 12515.217,E2 12515.217} C_VEL
LIN {X 0,Y 263.92,Z 1063.034,A -85,B 0,C 180,E1 12510.434,E2 12510.434} C_VEL
LIN {X 0,Y 263.91,Z 1062.353,A -85,B 0,C 180,E1 12505.872,E2 12505.872} C_VEL
LIN {X 0,Y 264.048,Z 1060.691,A -85,B 0,C 180,E1 12501.507,E2 12501.507} C_VEL
LIN {X 0,Y 264.572,Z 1058.016,A -85,B 0,C 180,E1 12497.116,E2 12497.116} C_VEL
LIN {X 0,Y 265.797,Z 1054.306,A -85,B 0,C 180,E1 12492.712,E2 12492.712} C_VEL
LIN {X 0,Y 268.187,Z 1049.019,A -85,B 0,C 180,E1 12487.879,E2 12487.879} C_VEL
LIN {X 0,Y 272.679,Z 1040.968,A -85,B 0,C 180,E1 12482.245,E2 12482.245} C_VEL
LIN {X 0,Y 277.8,Z 1032.913,A -85,B 0,C 180,E1 12477.762,E2 12477.762} C_VEL
LIN {X 0,Y 284.8,Z 1022.758,A -85,B 0,C 180,E1 12473.105,E2 12473.105} C_VEL
LIN {X 0,Y 293.634,Z 1010.277,A -85,B 0,C 180,E1 12468.517,E2 12468.517} C_VEL
LIN {X 0,Y 301.677,Z 999.042,A -85,B 0,C 180,E1 12465.092,E2 12465.092} C_VEL
LIN {X 0,Y 311.441,Z 985.336,A -85,B 0,C 180,E1 12461.579,E2 12461.579} C_VEL
LIN {X 0,Y 322.797,Z 968.793,A -85,B 0,C 180,E1 12458.114,E2 12458.114} C_VEL
LIN {X 0,Y 332.746,Z 953.648,A -85,B 0,C 180,E1 12455.478,E2 12455.478} C_VEL
LIN {X 0,Y 343.66,Z 936.231,A -85,B 0,C 180,E1 12452.924,E2 12452.924} C_VEL
LIN {X 0,Y 355.183,Z 916.273,A -85,B 0,C 180,E1 12450.523,E2 12450.523} C_VEL
LIN {X 0,Y 364.316,Z 899.23,A -85,B 0,C 180,E1 12448.8,E2 12448.8} C_VEL
LIN {X 0,Y 374.065,Z 879.565,A -85,B 0,C 180,E1 12447.112,E2 12447.112} C_VEL
LIN {X 0,Y 384.339,Z 856.39,A -85,B 0,C 180,E1 12445.479,E2 12445.479} C_VEL
LIN {X 0,Y 392.24,Z 836.367,A -85,B 0,C 180,E1 12444.311,E2 12444.311} C_VEL
LIN {X 0,Y 399.684,Z 815.214,A -85,B 0,C 180,E1 12443.283,E2 12443.283} C_VEL
LIN {X 0,Y 407.354,Z 789.493,A -85,B 0,C 180,E1 12442.275,E2 12442.275} C_VEL
LIN {X 0,Y 412.537,Z 768.603,A -85,B 0,C 180,E1 12441.619,E2 12441.619} C_VEL
LIN {X 0,Y 417.223,Z 745.745,A -85,B 0,C 180,E1 12441.052,E2 12441.052} C_VEL
LIN {X 0,Y 421.329,Z 717.817,A -85,B 0,C 180,E1 12440.514,E2 12440.514} C_VEL
LIN {X 0,Y 432.333,Z 594.497,A -85,B 0,C 180,E1 12438.588,E2 12438.588} C_VEL
LIN {X 0,Y 440.669,Z 500.991,A -85,B 0,C 180,E1 12437.156,E2 12437.156} C_VEL
LIN {X 0,Y 435.392,Z 491.502,A -85,B 0,C 180,E1 12434.429,E2 12434.429} C_VEL
LIN {X 0,Y 430.91,Z 483.755,A -85,B 0,C 180,E1 12431.647,E2 12431.647} C_VEL
LIN {X 0,Y 428.022,Z 478.999,A -85,B 0,C 180,E1 12429.479,E2 12429.479} C_VEL
LIN {X 0,Y 425.791,Z 475.211,A -85,B 0,C 180,E1 12427.421,E2 12427.421} C_VEL
LIN {X 0,Y 423.337,Z 470.924,A -85,B 0,C 180,E1 12424.335,E2 12424.335} C_VEL
LIN {X 0,Y 421.47,Z 467.798,A -85,B 0,C 180,E1 12418.505,E2 12418.505} C_VEL
LIN {X 0,Y 421.84,Z 469.136,A -85,B 0,C 180,E1 12415.514,E2 12415.514} C_VEL
LIN {X 0,Y 423.663,Z 471.443,A -85,B 0,C 180,E1 12411.996,E2 12411.996} C_VEL
LIN {X 0,Y 426.559,Z 476.474,A -85,B 0,C 180,E1 12408.644,E2 12408.644} C_VEL
LIN {X 0,Y 429.394,Z 481.263,A -85,B 0,C 180,E1 12406.26,E2 12406.26} C_VEL
LIN {X 0,Y 432.938,Z 487.29,A -85,B 0,C 180,E1 12403.841,E2 12403.841} C_VEL
LIN {X 0,Y 437.404,Z 495.011,A -85,B 0,C 180,E1 12401.3,E2 12401.3} C_VEL
LIN {X 0,Y 440.608,Z 501.144,A -85,B 0,C 180,E1 12399.681,E2 12399.681} C_VEL
LIN {X 0,Y 421.599,Z 714.079,A -85,B 0,C 180,E1 12396.387,E2 12396.387} C_VEL
LIN {X 0,Y 417.774,Z 740.883,A -85,B 0,C 180,E1 12395.875,E2 12395.875} C_VEL
LIN {X 0,Y 412.94,Z 764.782,A -85,B 0,C 180,E1 12395.277,E2 12395.277} C_VEL
LIN {X 0,Y 407.571,Z 786.643,A -85,B 0,C 180,E1 12394.575,E2 12394.575} C_VEL
LIN {X 0,Y 399.863,Z 812.538,A -85,B 0,C 180,E1 12393.534,E2 12393.534} C_VEL
LIN {X 0,Y 392.751,Z 832.86,A -85,B 0,C 180,E1 12392.527,E2 12392.527} C_VEL
LIN {X 0,Y 385.025,Z 852.495,A -85,B 0,C 180,E1 12391.374,E2 12391.374} C_VEL
LIN {X 0,Y 374.659,Z 875.966,A -85,B 0,C 180,E1 12389.708,E2 12389.708} C_VEL
LIN {X 0,Y 364.894,Z 895.665,A -85,B 0,C 180,E1 12388.005,E2 12388.005} C_VEL
LIN {X 0,Y 355.158,Z 913.786,A -85,B 0,C 180,E1 12386.152,E2 12386.152} C_VEL
LIN {X 0,Y 342.644,Z 935.122,A -85,B 0,C 180,E1 12383.509,E2 12383.509} C_VEL
LIN {X 0,Y 332.635,Z 950.995,A -85,B 0,C 180,E1 12381.127,E2 12381.127} C_VEL
LIN {X 0,Y 321.284,Z 968.174,A -85,B 0,C 180,E1 12378.056,E2 12378.056} C_VEL
LIN {X 0,Y 310.16,Z 983.983,A -85,B 0,C 180,E1 12374.564,E2 12374.564} C_VEL
LIN {X 0,Y 301.345,Z 996.255,A -85,B 0,C 180,E1 12371.322,E2 12371.322} C_VEL
LIN {X 0,Y 291.734,Z 1009.557,A -85,B 0,C 180,E1 12367.101,E2 12367.101} C_VEL
LIN {X 0,Y 283.564,Z 1020.809,A -85,B 0,C 180,E1 12362.649,E2 12362.649} C_VEL
LIN {X 0,Y 277.42,Z 1029.681,A -85,B 0,C 180,E1 12358.409,E2 12358.409} C_VEL
LIN {X 0,Y 271.564,Z 1038.85,A -85,B 0,C 180,E1 12352.972,E2 12352.972} C_VEL
LIN {X 0,Y 267.93,Z 1045.313,A -85,B 0,C 180,E1 12348.044,E2 12348.044} C_VEL
LIN {X 0,Y 265.787,Z 1050.032,A -85,B 0,C 180,E1 12343.488,E2 12343.488} C_VEL
LIN {X 0,Y 264.412,Z 1054.259,A -85,B 0,C 180,E1 12338.043,E2 12338.043} C_VEL
LIN {X 0,Y 263.976,Z 1056.619,A -85,B 0,C 180,E1 12333.04,E2 12333.04} C_VEL
LIN {X 0,Y 263.914,Z 1057.65,A -85,B 0,C 180,E1 12328.914,E2 12328.914} C_VEL
LIN {X 0,Y 263.917,Z 1057.803,A -85,B 0,C 180,E1 12324.783,E2 12324.783} C_VEL
LIN {X 0,Y 264.001,Z 1057.074,A -85,B 0,C 180,E1 12320.627,E2 12320.627} C_VEL
LIN {X 0,Y 264.362,Z 1055.444,A -85,B 0,C 180,E1 12316.421,E2 12316.421} C_VEL
LIN {X 0,Y 265.334,Z 1052.763,A -85,B 0,C 180,E1 12312,E2 12312} C_VEL
LIN {X 0,Y 267.25,Z 1048.843,A -85,B 0,C 180,E1 12307.334,E2 12307.334} C_VEL
LIN {X 0,Y 271.24,Z 1042.358,A -85,B 0,C 180,E1 12301.606,E2 12301.606} C_VEL
LIN {X 0,Y 276.343,Z 1035.054,A -85,B 0,C 180,E1 12296.702,E2 12296.702} C_VEL
LIN {X 0,Y 282.552,Z 1026.882,A -85,B 0,C 180,E1 12292.251,E2 12292.251} C_VEL
LIN {X 0,Y 292.038,Z 1014.875,A -85,B 0,C 180,E1 12287.052,E2 12287.052} C_VEL
LIN {X 0,Y 300.724,Z 1004.017,A -85,B 0,C 180,E1 12283.268,E2 12283.268} C_VEL
LIN {X 0,Y 311.595,Z 990.405,A -85,B 0,C 180,E1 12279.344,E2 12279.344} C_VEL
LIN {X 0,Y 323.13,Z 975.217,A -85,B 0,C 180,E1 12275.833,E2 12275.833} C_VEL
LIN {X 0,Y 333.272,Z 961.398,A -85,B 0,C 180,E1 12273.169,E2 12273.169} C_VEL
LIN {X 0,Y 345.547,Z 943.852,A -85,B 0,C 180,E1 12270.342,E2 12270.342} C_VEL
LIN {X 0,Y 357.524,Z 925.192,A -85,B 0,C 180,E1 12267.901,E2 12267.901} C_VEL
LIN {X 0,Y 367.768,Z 908.133,A -85,B 0,C 180,E1 12266.03,E2 12266.03} C_VEL
LIN {X 0,Y 379.453,Z 886.934,A -85,B 0,C 180,E1 12264.088,E2 12264.088} C_VEL
LIN {X 0,Y 389.31,Z 866.951,A -85,B 0,C 180,E1 12262.583,E2 12262.583} C_VEL
LIN {X 0,Y 397.417,Z 848.842,A -85,B 0,C 180,E1 12261.424,E2 12261.424} C_VEL
LIN {X 0,Y 406.884,Z 825.248,A -85,B 0,C 180,E1 12260.16,E2 12260.16} C_VEL
LIN {X 0,Y 414.904,Z 801.554,A -85,B 0,C 180,E1 12259.146,E2 12259.146} C_VEL
LIN {X 0,Y 421.074,Z 780.434,A -85,B 0,C 180,E1 12258.411,E2 12258.411} C_VEL
LIN {X 0,Y 427.133,Z 755.479,A -85,B 0,C 180,E1 12257.713,E2 12257.713} C_VEL
LIN {X 0,Y 428.247,Z 749.751,A -85,B 0,C 180,E1 12257.582,E2 12257.582} C_VEL
LIN {X 0,Y 429.406,Z 742.364,A -85,B 0,C 180,E1 12257.3,E2 12257.3} C_VEL
LIN {X 0,Y 430.634,Z 723.058,A -85,B 0,C 180,E1 12256.131,E2 12256.131} C_VEL
LIN {X 0,Y 431.2,Z 716.612,A -85,B 0,C 180,E1 12255.925,E2 12255.925} C_VEL
LIN {X 0,Y 437.967,Z 647.543,A -85,B 0,C 180,E1 12254.873,E2 12254.873} C_VEL
LIN {X 0,Y 450.573,Z 515.41,A -85,B 0,C 180,E1 12252.893,E2 12252.893} C_VEL
LIN {X 0,Y 447.266,Z 509.305,A -85,B 0,C 180,E1 12250.693,E2 12250.693} C_VEL
LIN {X 0,Y 444.859,Z 505.035,A -85,B 0,C 180,E1 12248.792,E2 12248.792} C_VEL
LIN {X 0,Y 443.363,Z 502.266,A -85,B 0,C 180,E1 12247.386,E2 12247.386} C_VEL
LIN {X 0,Y 441.294,Z 498.473,A -85,B 0,C 180,E1 12244.939,E2 12244.939} C_VEL
LIN {X 0,Y 439.342,Z 494.076,A -85,B 0,C 180,E1 12240.522,E2 12240.522} C_VEL
LIN {X 0,Y 439.425,Z 494.237,A -85,B 0,C 180,E1 12236.216,E2 12236.216} C_VEL
LIN {X 0,Y 441.265,Z 498.504,A -85,B 0,C 180,E1 12232.186,E2 12232.186} C_VEL
LIN {X 0,Y 442.005,Z 499.795,A -85,B 0,C 180,E1 12231.217,E2 12231.217} C_VEL
LIN {X 0,Y 444.263,Z 503.892,A -85,B 0,C 180,E1 12228.839,E2 12228.839} C_VEL
LIN {X 0,Y 447.067,Z 508.908,A -85,B 0,C 180,E1 12226.55,E2 12226.55} C_VEL
LIN {X 0,Y 450.641,Z 515.653,A -85,B 0,C 180,E1 12224.152,E2 12224.152} C_VEL
LIN {X 0,Y 431.279,Z 716.943,A -85,B 0,C 180,E1 12221.14,E2 12221.14} C_VEL
LIN {X 0,Y 427.19,Z 743.889,A -85,B 0,C 180,E1 12220.658,E2 12220.658} C_VEL
LIN {X 0,Y 422.112,Z 767.578,A -85,B 0,C 180,E1 12220.119,E2 12220.119} C_VEL
LIN {X 0,Y 416.942,Z 787.396,A -85,B 0,C 180,E1 12219.557,E2 12219.557} C_VEL
LIN {X 0,Y 409.497,Z 811.629,A -85,B 0,C 180,E1 12218.706,E2 12218.706} C_VEL
LIN {X 0,Y 400.592,Z 835.636,A -85,B 0,C 180,E1 12217.634,E2 12217.634} C_VEL
LIN {X 0,Y 392.327,Z 855.383,A -85,B 0,C 180,E1 12216.563,E2 12216.563} C_VEL
LIN {X 0,Y 382.063,Z 877.334,A -85,B 0,C 180,E1 12215.138,E2 12215.138} C_VEL
LIN {X 0,Y 370.997,Z 898.171,A -85,B 0,C 180,E1 12213.481,E2 12213.481} C_VEL
LIN {X 0,Y 360.777,Z 915.863,A -85,B 0,C 180,E1 12211.803,E2 12211.803} C_VEL
LIN {X 0,Y 348.137,Z 936.047,A -85,B 0,C 180,E1 12209.5,E2 12209.5} C_VEL
